REGION Network 8: Reset Counters
   RUNG wire#powerrail
      Contact( #Reset_Counters )
      Move(in := 0, out1 => "DB_STATUS_IJCORE".AW_number)
      Move(in := T#0MS, out1 => "DB_STATUS_IJCORE".AW_durationMax)
   END_RUNG
   // the same network as SCL:
   IF #Reset_Counters THEN
       "DB_STATUS_IJCORE".AW_number := 0;
       "DB_STATUS_IJCORE".AW_durationMax := T#0MS;
   END_IF;
END_REGION
END_FUNCTION_BLOCK

FUNCTION_BLOCK "IJC PROTOCOL"
{ S7_Optimized_Access := 'TRUE' }
AUTHOR : RAUL_ROBINS
VERSION : 0.1
   VAR_INPUT RETAIN
      M_TYPE : String[3];
      M_NBR : DInt;
   END_VAR
   VAR_INPUT 
      DB_REC : DB_ANY;
      DB_SEND : DB_ANY;
      START_MSG : Bool;
      KANBAN : String[30];
      SAP_PN : String[16];
      COMPONENT : String[64];
      START_SCREW : Bool;
      "SCREW T_INT" : Word;
      "SCREW T_FLOAT" : Word;
      "SCREW ANGLE" : Word;
      ERR_RESET : Bool;
      PROCESS_STATUS { ExternalAccessible := 'False'; ExternalVisible := 'False'; ExternalWritable := 'False'} : SInt;
      NUM_OF_PROCESS : SInt;
   END_VAR

   VAR_OUTPUT 
      SEQ_STEP : Int;
      DN : Bool;
      FLT : Bool;
      ANS : SInt;
      A_TMOUT : Bool;
      M_TMOUT : Bool;
      NFP : String[8];
   END_VAR

   VAR_IN_OUT 
      AWAKE_SW : Int;
   END_VAR

   VAR 
      MSG_TMOUT {InstructionName := 'TON_TIME'; LibVersion := '1.0'} : TON_TIME;
      AWK_TMR {InstructionName := 'TON_TIME'; LibVersion := '1.0'} : TON_TIME;
      AWK_TMOUT {InstructionName := 'TON_TIME'; LibVersion := '1.0'} : TON_TIME;
      "SCREW NBR" { S7_SetPoint := 'True'} : Word;
      SCREW : Array[1..9] of Struct
         ANGLE : Word;
         TORQUE : Struct
            "INT" : Word;
            FLOAT : Word;
         END_STRUCT;
      END_STRUCT;
      HMI : Struct
         SEND : Struct
            MSG : String[50];
            SW : SInt;
         END_STRUCT;
         RCV : Struct
            MSG : String[50];
            SW : SInt;
         END_STRUCT;
      END_STRUCT;
      ONS : Array[1..10] of Bool;
   END_VAR

   VAR_TEMP 
      MSG_TYPE : SInt;
      IDB : Int;
      i : Int;
      j : Int;
      k : Int;
      SEND_OFFSET : Struct
         SW : DInt;
         MSG : DInt;
      END_STRUCT;
      REC_OFFSET : Struct
         SW : DInt;
         ANS : DInt;
         MSG : DInt;
      END_STRUCT;
      CNT : SInt;
      CNT_STR : String[2];
      TMP : Word;
      BTEST : Bool;
      STATUS : Char;
      NUMBER : Char;
      CHAR_ARRAY : Array[0..49] of Char;
   END_VAR

   VAR CONSTANT 
      "DB" : Byte := 16#84;
      CLEAR : Word := 16#0;
      MINUS1 : Word := 16#FFFF;
      PLUS1 : Word := 16#1;
   END_VAR


BEGIN
	(*     IJCORE PROTOCOL
	CREATED BY: RAUL ROBINS
	CREATED ON: 08/05/2020
	VERSION: 1.0
	*)
	
	//***** CLEAR ALL FAULTS ***************************************
	IF #ERR_RESET OR
	NOT #START_MSG THEN
	    #M_TMOUT := false;
	    #FLT := FALSE;
	END_IF;
	
	//***** AWAKE SIGNAL ***************************************
	  //#AWK_TMR(IN := (#AWAKE_SW <= 0),
	  //      PT := T#500ms);
	
	//IF #AWK_TMR.Q AND
	  //  #AWAKE_SW <= 1 THEN
	   // #AWAKE_SW := 1;
	//END_IF;
	
	
	//AWAKE TIMEOUT
	//#AWK_TMOUT(IN := (#AWAKE_SW = 1),
	  //      PT := T#6S);
	//IF #AWK_TMOUT.Q THEN
	    //#A_TMOUT := TRUE;
	//ELSIF (#AWAKE_SW < 0) THEN
	  //  #A_TMOUT := FALSE;
	//END_IF;
	
	// ***** TIMEOUT FOR ANSWER FROM IJC **********************************
	// WAITMOUNT FOR FAULT
	// 
	#MSG_TMOUT(IN := (#SEQ_STEP = 50 OR #SEQ_STEP = 60),
	           PT := T#60S,
	           Q => #BTEST);
	//SET FAULT
	 IF #MSG_TMOUT.Q THEN
	     #M_TMOUT := true;
	     #SEQ_STEP := 0;
	END_IF;
	
	//***** VALID MESSAGE NUMBER ***************************************
	IF #M_NBR < 1 THEN
	    RETURN;
	END_IF;
	
	//***** MESSAGE TYPE SELECTED ***************************************
	IF    #M_TYPE = 'CNF' THEN
	    #MSG_TYPE := 1;
	ELSIF #M_TYPE = 'TRC' THEN
	    #MSG_TYPE := 1;
	ELSIF #M_TYPE = 'TRB' THEN
	    #MSG_TYPE := 1;
	ELSIF #M_TYPE = 'TRS' THEN
	    #MSG_TYPE := 2;
	ELSIF #M_TYPE = 'TRI' THEN
	    #MSG_TYPE := 3;
	ELSIF #M_TYPE = 'TRE' THEN
	    #MSG_TYPE := 4;
	ELSIF #M_TYPE = 'STA' THEN
	    #MSG_TYPE := 5;
	ELSIF #M_TYPE = 'CMA' THEN
	    #MSG_TYPE := 6;
	ELSIF #M_TYPE = 'TRR' THEN
	    #MSG_TYPE := 7;
	ELSIF #M_TYPE = 'TRW' THEN
	    #MSG_TYPE := 8;
	ELSIF #M_TYPE = 'PFC' THEN
	    #MSG_TYPE := 9;
	ELSIF #M_TYPE = 'NFP' THEN
	    #MSG_TYPE := 10;
	ELSE
	    RETURN;
	END_IF;
	
	//***** MESSAGE OFFSET CALC ***************************************
	#SEND_OFFSET.SW := (#M_NBR * 2) + 2;
	#SEND_OFFSET.MSG := ((#M_NBR - 1) * 80) + 604;
	#REC_OFFSET.SW := (#M_NBR - 1) * 2;
	#REC_OFFSET.ANS := ((#M_NBR - 1) * 32) + 600;
	#REC_OFFSET.MSG := ((#M_NBR - 1) * 32) + 602;
	#HMI.SEND.SW := WORD_TO_SINT(PEEK_WORD(area := #DB, dbNumber := #DB_SEND, byteOffset := #SEND_OFFSET.SW));
	#HMI.RCV.SW := WORD_TO_SINT(PEEK_WORD(area := #DB, dbNumber := #DB_REC, byteOffset := #REC_OFFSET.SW));
	
	//***** GET SCREW DATA ***************************************
	
	//CLEAR SCREW DATA*************************************************
	// IF NOT #START_SCREW THEN
	//     #"SCREW NBR" := 0;
	//     FOR #i := 1 TO 9 BY 1 DO
	//         #SCREW[#i].TORQUE."INT" := 0;
	//         #SCREW[#i].TORQUE.FLOAT := 0;
	//         #SCREW[#i].ANGLE := 0;
	//     END_FOR;
	// END_IF;
	
	// IF  #START_SCREW   AND
	//     #"SCREW ANGLE" > 0 AND
	//     #"SCREW NBR"< 9 THEN
	//     IF NOT #ONS[2] THEN
	//         #"SCREW NBR" += 1;
	//         #SCREW[#"SCREW NBR"].TORQUE."INT" := #"SCREW T_INT";
	//         #SCREW[#"SCREW NBR"].TORQUE.FLOAT := #"SCREW T_FLOAT";
	//         #SCREW[#"SCREW NBR"].ANGLE := #"SCREW ANGLE";
	// //ONE SHOT
	//         #ONS[2] := True;
	//     END_IF;
	// ELSE
	//     #ONS[2] := False;
	// END_IF;
	#"SCREW NBR" := SINT_TO_WORD(#NUM_OF_PROCESS);
	
	
	////////////////////////////////////////////////////////////////////
	//START IJCORE SEQUENCE
	//>>>>>STEP-00 ->>>>>>>>>>>>>>>>>>>>>>>>>>>>>>>>>>>>>>>>>>>>>>>>>>>>>
	//WAIT FLAG SEND TO START SEQUENCE
	
	IF  NOT #START_MSG THEN
	    #DN := FALSE;
	    #SEQ_STEP := 0;
	    #ANS := 0;
	    //MESSAGE
	    FOR #i := 0 TO 79 DO
	        POKE(area := #DB,
	             dbNumber := #DB_SEND,
	             byteOffset := (#SEND_OFFSET.MSG + #i),
	             value := ' ');
	    END_FOR;
	    //SW_MESSAGE
	    POKE(area := #DB,
	         dbNumber := #DB_SEND,
	         byteOffset := #SEND_OFFSET.SW,
	         value := #CLEAR);
	ELSE
	    //***** HMI SIGNAL STATUS ***************************************
	    //SEND
	    FOR #i := 0 TO 49 BY 1 DO
	        #CHAR_ARRAY[#i] := BYTE_TO_CHAR(PEEK(area := #DB, dbNumber := #DB_SEND, byteOffset := #SEND_OFFSET.MSG + #i));
	    END_FOR;
	    
	    Chars_TO_Strg(Chars := #CHAR_ARRAY,
	                  pChars := 0,
	                  Cnt := 50,
	                  Strg => #HMI.SEND.MSG);
	    
	    
	    //NFP
	    //
	    
	    // #NFP := '';
	
	    // RETURN;
	END_IF;
	
	
	//***** HMI SIGNAL STATUS ***************************************
	//SEND
	//FOR #i := 0 TO 49 BY 1 DO
	  //  #CHAR_ARRAY[#i] := BYTE_TO_CHAR(PEEK(area := #DB, dbNumber := #DB_SEND, byteOffset := #SEND_OFFSET.MSG + #i));
	//END_FOR;
	
	//Chars_TO_Strg(Chars := #CHAR_ARRAY,
	  //            pChars := 0,
	    //          #CNT := 50,
	      //        Strg => #HMI.SEND.MSG);
	
	
	//HMI REC
	FOR #i := 0 TO 49 BY 1 DO
	    #CHAR_ARRAY[#i] := BYTE_TO_CHAR(PEEK(area := #DB, dbNumber := #DB_REC, byteOffset := #REC_OFFSET.MSG + #i));
	END_FOR;
	
	Chars_TO_Strg(Chars := #CHAR_ARRAY,
	              pChars := 0,
	              Cnt := 50,
	              Strg => #HMI.RCV.MSG);
	
	//***** START SEQUENCE ***************************************
	IF #SEQ_STEP = 0 AND #SEQ_STEP<>100 AND 
	    #START_MSG THEN
	    #SEQ_STEP := 10;
	END_IF;
	
	//>>>>>STEP-10 ->>>>>>>>>>>>>>>>>>>>>>>>>>>>>>>>>>>>>>>>>>>>>>>>>>>>>
	//TURN OFF SEND FLAG
	IF #SEQ_STEP = 10 AND #SEQ_STEP<>100 AND  #START_MSG THEN
	    //GOTO STEP 30
	    #SEQ_STEP := 30;
	END_IF;
	
	//>>>>>STEP-30 ->>>>>>>>>>>>>>>>>>>>>>>>>>>>>>>>>>>>>>>>>>>>>>>>>>>>>
	//INIT DATA DB5 or DB1005 
	IF #SEQ_STEP = 30 THEN
	    //SET FLAGS TO 0
	    POKE(area := #DB,
	         dbNumber := #DB_SEND,
	         byteOffset := #SEND_OFFSET.SW,
	         value := #CLEAR);
	    POKE(area := #DB,
	         dbNumber := #DB_REC,
	         byteOffset := #REC_OFFSET.SW,
	         value := #CLEAR);
	    POKE(area := #DB,
	         dbNumber := #DB_REC,
	         byteOffset := #REC_OFFSET.ANS,
	         value := #CLEAR);
	    
	    //CLEAR DBSEND MESSAGE
	    FOR #i := 0 TO 79 BY 1 DO
	        POKE(area := #DB,
	             dbNumber := #DB_SEND,
	             byteOffset := (#SEND_OFFSET.MSG + #i),
	             value := ' ');
	    END_FOR;
	    FOR #i := 0 TO 69 BY 1 DO
	        POKE(area := #DB,
	             dbNumber := #DB_REC,
	             byteOffset := (#REC_OFFSET.MSG + #i),
	             value := ' ');
	    END_FOR;
	    //GO TO STEP 40
	    #SEQ_STEP := 40;
	END_IF;
	
	//>>>>>STEP-40 ->>>>>>>>>>>>>>>>>>>>>>>>>>>>>>>>>>>>>>>>>>>>>>>>>>>>>
	//CREATE MESSAGE
	IF #SEQ_STEP = 40 THEN
	    //MESSAGE TYPE
	   
	    //COPY KANBAN
	    FOR #i := 0 TO 7 BY 1 DO
	        POKE(area := #DB,
	             dbNumber := #DB_SEND,
	             byteOffset := (#SEND_OFFSET.MSG + #i),
	             value := #KANBAN[#i+1]);
	    END_FOR;
	    
	    //CONVERT DATATYPE
	    #STATUS := SINT_TO_CHAR(#PROCESS_STATUS + 48);
	    #NUMBER := SINT_TO_CHAR(#NUM_OF_PROCESS + 48);
	    
	    CASE #MSG_TYPE OF
	        1://CNF & TRC
	            #CNT := INT_TO_SINT (LEN(#COMPONENT));
	            VAL_STRG(IN := #CNT,
	                     SIZE := 2,
	                     PREC := 0,
	                     FORMAT := W#16#0,
	                     P := 1,
	                     OUT => #CNT_STR);
	            IF #CNT < 10 THEN
	                #CNT_STR := REPLACE(IN1 := #CNT_STR, IN2 := '0',
	                                    L := 1,
	                                    P := FIND(IN1 := #CNT_STR,
	                                              IN2 := ' '));
	            END_IF;
	            POKE(area := #DB,
	                 dbNumber := #DB_SEND,
	                 byteOffset := (#SEND_OFFSET.MSG + 8),
	                 value := #CNT_STR[1]);
	            POKE(area := #DB,
	                 dbNumber := #DB_SEND,
	                 byteOffset := (#SEND_OFFSET.MSG + 9),
	                 value := #CNT_STR[2]);
	            FOR #i := 0 TO 28 BY 1 DO
	                POKE(area := #DB,
	                     dbNumber := #DB_SEND,
	                     byteOffset := (#SEND_OFFSET.MSG + #i + 10),
	                     value := #COMPONENT[#i+1]);
	            END_FOR;
	            
	        2://TRS
	            #NUMBER := WORD_TO_CHAR(#"SCREW NBR" + 48);
	            POKE(area := #DB,
	                 dbNumber := #DB_SEND,
	                 byteOffset := (#SEND_OFFSET.MSG + 8),
	                 value := #STATUS);
	            POKE(area := #DB,
	                 dbNumber := #DB_SEND,
	                 byteOffset := (#SEND_OFFSET.MSG + 9),
	                 value := #NUMBER);
	            FOR #i := 0 TO 8 BY 1 DO
	                #j := #i + 1;
	                #k := (#i * 6) + 10;
	                //ANGLE
	                POKE(area := #DB,
	                     dbNumber := #DB_SEND,
	                     byteOffset := (#SEND_OFFSET.MSG + #k ),
	                     value :=  #SCREW[#j].ANGLE);
	                //TORQUE BEFORE POINT
	                POKE(area := #DB,
	                     dbNumber := #DB_SEND,
	                     byteOffset := (#SEND_OFFSET.MSG + #k + 2),
	                     value := #SCREW[#j].TORQUE."INT");
	        
	                //TORQUE AFTER POINT
	                POKE(area := #DB,
	                     dbNumber := #DB_SEND,
	                     byteOffset := (#SEND_OFFSET.MSG + #k + 4),
	                     value := #SCREW[#j].TORQUE."FLOAT");
	            END_FOR;
	            
	        3://TRI
	            POKE(area := #DB,
	                 dbNumber := #DB_SEND,
	                 byteOffset := (#SEND_OFFSET.MSG + 8),
	                 value := #STATUS);
	        4://TRE 
	            POKE(area := #DB,
	                 dbNumber := #DB_SEND,
	                 byteOffset := (#SEND_OFFSET.MSG + 8),
	                 value := '9');;
	            POKE(area := #DB,
	                 dbNumber := #DB_SEND,
	                 byteOffset := (#SEND_OFFSET.MSG + 9),     
	                 value := '9');                                 
	            POKE(area := #DB,
	                 dbNumber := #DB_SEND,
	                 byteOffset := (#SEND_OFFSET.MSG + 10),
	                 value := #STATUS);
	        5://STA
	            ;
	        6://TRB
	            POKE(area := #DB,
	                 dbNumber := #DB_SEND,
	                 byteOffset := (#SEND_OFFSET.MSG + 9),
	                 value := '1');;
	            POKE(area := #DB,
	                 dbNumber := #DB_SEND,
	                 byteOffset := (#SEND_OFFSET.MSG + 10),
	                 value := '6');
	            FOR #i := 1 TO 16 BY 1 DO
	                POKE(area := #DB,
	                     dbNumber := #DB_SEND,
	                     byteOffset := (#SEND_OFFSET.MSG + #i + 1),
	                     value := #SAP_PN[#i]);
	            END_FOR;
	            ;
	        7://TRR
	            POKE(area := #DB,
	                 dbNumber := #DB_SEND,
	                 byteOffset := (#SEND_OFFSET.MSG + 8),
	                 value := #STATUS);
	            POKE(area := #DB,
	                 dbNumber := #DB_SEND,
	                 byteOffset := (#SEND_OFFSET.MSG + 9),
	                 value := #NUMBER);
	            
	        8://TRW
	            POKE(area := #DB,
	                 dbNumber := #DB_SEND,
	                 byteOffset := (#SEND_OFFSET.MSG + 8),
	                 value := #STATUS);
	            POKE(area := #DB,
	                 dbNumber := #DB_SEND,
	                 byteOffset := (#SEND_OFFSET.MSG + 9),
	                 value := #NUMBER);
	            
	        9://PFC
	            #CNT := INT_TO_SINT(LEN(#COMPONENT));
	            VAL_STRG(IN := #CNT,
	                     SIZE := 2,
	                     PREC := 0,
	                     FORMAT := W#16#0,
	                     P := 1,
	                     OUT => #CNT_STR);
	            IF #CNT < 10 THEN
	                #CNT_STR := REPLACE(IN1 := #CNT_STR, IN2 := '0',
	                                    L := 1,
	                                    P := FIND(IN1 := #CNT_STR,
	                                              IN2 := ' '));
	            END_IF;
	            POKE(area := #DB,
	                 dbNumber := #DB_SEND,
	                 byteOffset := (#SEND_OFFSET.MSG + 8),
	                 value := #CNT_STR[1]);
	            POKE(area := #DB,
	                 dbNumber := #DB_SEND,
	                 byteOffset := (#SEND_OFFSET.MSG + 9),
	                 value := #CNT_STR[2]);
	            FOR #i := 0 TO 28 BY 1 DO
	                POKE(area := #DB,
	                     dbNumber := #DB_SEND,
	                     byteOffset := (#SEND_OFFSET.MSG + #i + 10),
	                     value := #COMPONENT[#i + 1]);
	            END_FOR;
	        10://NFP
	            POKE(area := #DB,
	                 dbNumber := #DB_SEND,
	                 byteOffset := (#SEND_OFFSET.MSG),
	                 value := '0');
	            POKE(area := #DB,
	                 dbNumber := #DB_SEND,
	                 byteOffset := (#SEND_OFFSET.MSG + 1),
	                 value := '8');
	            FOR #i := 1 TO 8 BY 1 DO
	                POKE(area := #DB,
	                     dbNumber := #DB_SEND,
	                     byteOffset := (#SEND_OFFSET.MSG + #i + 1),
	                     value := #KANBAN[#i]);
	            END_FOR;
	    END_CASE;
	    
	    //SET FLAG TO I TO INFORM THAT PLC IS READY (DB5 Ó 1005)
	    POKE(area := #DB,
	         dbNumber := #DB_SEND,
	         byteOffset := #SEND_OFFSET.SW,
	         value := #PLUS1);
	   #SEQ_STEP := 50;
	END_IF;
	
	//***** WAIT ANSWER FROM IJC***** **********************************
	//CHECK FLAG IN STEP-50
	IF #SEQ_STEP = 50 THEN
	    //WAIT FOR SEND FLAG TO BE -1
	    IF PEEK_WORD(area := #DB, dbNumber := #DB_SEND, byteOffset := #SEND_OFFSET.SW) = #MINUS1 THEN
	        #SEQ_STEP := 60;//GO TO STEP 60
	    END_IF;
	END_IF;
	
	//>>>>>STEP-60 ->>>>>>>>>>>>>>>>>>>>>>>>>>>>>>>>>>>>>>>>>>>>>>>>>>>>>
	//COPY NFP MESSAGE TO LOCAL IJC_DB AND ANSWER -1 TO IJC
	IF #SEQ_STEP = 60 THEN
	    //POINTER OFFSET TO STATUS WORD
	    IF PEEK_WORD(area := #DB, dbNumber := #DB_REC, byteOffset := #REC_OFFSET.SW) = #PLUS1 THEN
	        #ANS := (PEEK_WORD(area := #DB, dbNumber := #DB_REC, byteOffset := #REC_OFFSET.ANS));
	        #TMP := (PEEK_WORD(area := #DB, dbNumber := #DB_REC, byteOffset := #REC_OFFSET.ANS));
	     //COPY NFP RECEIVED
	        FOR #i := 0 TO 7 BY 1 DO
	            #CHAR_ARRAY[#i] := PEEK_BYTE(area := #DB, dbNumber := #DB_REC, byteOffset := #REC_OFFSET.MSG+#i);
	        END_FOR;
	        Chars_TO_Strg(Chars:=#CHAR_ARRAY,
	                      pChars:=0,
	                      Cnt:=8,
	                      Strg=>#NFP);
	        //SET TO -1 REC
	        POKE(area := #DB,
	             dbNumber := #DB_REC,
	             byteOffset := #REC_OFFSET.SW,
	             value := #MINUS1);
	        #DN := TRUE;
	        #SEQ_STEP := 100;
	    END_IF;
	END_IF;
	
	
	IF #TMP < 0 THEN
	    #FLT := TRUE;
	END_IF;
	//RESET FAULT
	
	
	//***** END**********************************************************************
	
END_FUNCTION_BLOCK

FUNCTION_BLOCK "IJCoreMain"   // FB1000, LAD
TITLE = IJCore Main
{ S7_Optimized_Access := 'TRUE' }
VERSION : 0.1
// stored: AutoNumber false, IsIECCheckEnabled false, IsRetainMemResEnabled false, MemoryReserve 100, SetENOAutomatically false, UDAEnableTagReadback false
   VAR
      Enable : Bool;
      Mode : UInt;
      Indicator : Int;
      AlarmReset : Bool;
      AWAKE_SIGNAL { S7_SetPoint := 'True'} : "AWAKE_SIGNAL";
      MSG : Array[1..20] of "IJCoreMessageProcotol";
      NFP { S7_SetPoint := 'True'} : Array[1..4] of String[30];
   END_VAR
   VAR_TEMP
      MessageDone : Bool;
      Answer : DInt;
      Fault : DInt;
   END_VAR
   VAR CONSTANT
      STA : Int := 5;
      CNF : Int := 1;
      TRC : Int := 13;
      PFC : Int := 9;
      TRR : Int := 7;
   END_VAR
BEGIN

REGION Network 1
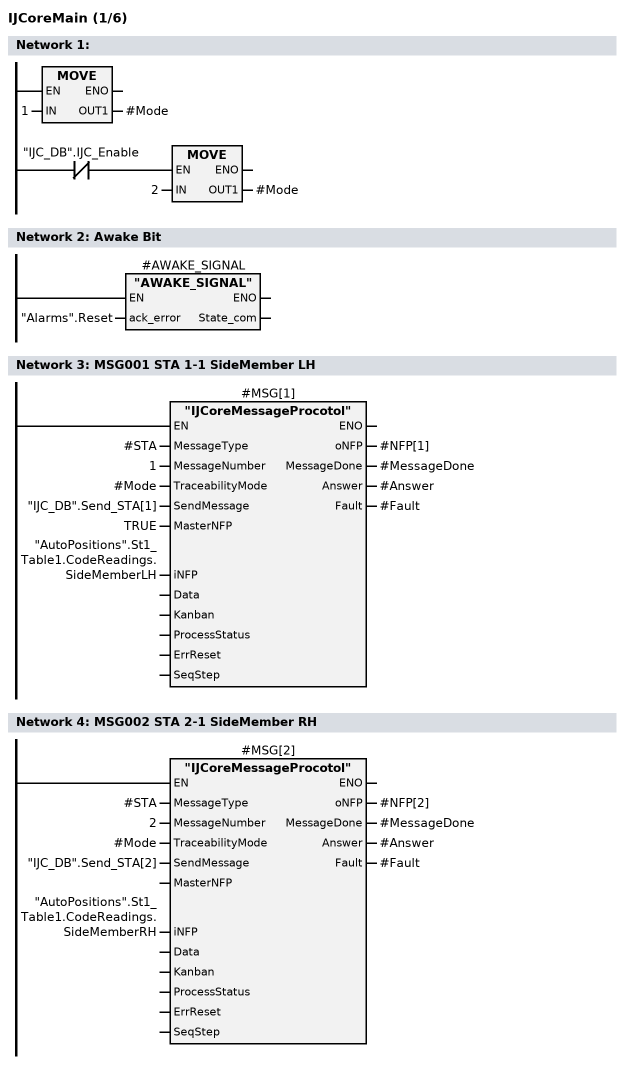
   RUNG wire#powerrail
      Move(in := 1, out1 => #Mode)
   END_RUNG
   RUNG wire#powerrail
      I_Contact( "IJC_DB".IJC_Enable )
      Move(in := 2, out1 => #Mode)
   END_RUNG
   // the same network as SCL:
   #Mode := 1;
   IF NOT "IJC_DB".IJC_Enable THEN #Mode := 2; END_IF;
END_REGION

REGION Network 2: Awake Bit
   RUNG wire#powerrail
      #AWAKE_SIGNAL(ack_error := "Alarms".Reset, State_com =>)
   END_RUNG
   // the same network as SCL:
   #AWAKE_SIGNAL(ack_error := "Alarms".Reset);   // "AWAKE_SIGNAL"
END_REGION

REGION Network 3: MSG001 STA 1-1 SideMember LH
   RUNG wire#powerrail
      #MSG[1](MessageType := #STA, MessageNumber := 1, TraceabilityMode := #Mode, SendMessage := "IJC_DB".Send_STA[1], MasterNFP := TRUE, iNFP := "AutoPositions".St1_Table1.CodeReadings.SideMemberLH, Data :=, Kanban :=, ProcessStatus :=, ErrReset :=, SeqStep :=, oNFP => #NFP[1], MessageDone => #MessageDone, Answer => #Answer, Fault => #Fault)
   END_RUNG
   // the same network as SCL:
   #MSG[1](MessageType := #STA,   // "IJCoreMessageProcotol"
           MessageNumber := 1,
           TraceabilityMode := #Mode,
           SendMessage := "IJC_DB".Send_STA[1],
           MasterNFP := TRUE,
           iNFP := "AutoPositions".St1_Table1.CodeReadings.SideMemberLH,
           oNFP => #NFP[1],
           MessageDone => #MessageDone,
           Answer => #Answer,
           Fault => #Fault);
END_REGION

REGION Network 4: MSG002 STA 2-1 SideMember RH
   RUNG wire#powerrail
      #MSG[2](MessageType := #STA, MessageNumber := 2, TraceabilityMode := #Mode, SendMessage := "IJC_DB".Send_STA[2], MasterNFP :=, iNFP := "AutoPositions".St1_Table1.CodeReadings.SideMemberRH, Data :=, Kanban :=, ProcessStatus :=, ErrReset :=, SeqStep :=, oNFP => #NFP[2], MessageDone => #MessageDone, Answer => #Answer, Fault => #Fault)
   END_RUNG
   // the same network as SCL:
   #MSG[2](MessageType := #STA,   // "IJCoreMessageProcotol"
           MessageNumber := 2,
           TraceabilityMode := #Mode,
           SendMessage := "IJC_DB".Send_STA[2],
           iNFP := "AutoPositions".St1_Table1.CodeReadings.SideMemberRH,
           oNFP => #NFP[2],
           MessageDone => #MessageDone,
           Answer => #Answer,
           Fault => #Fault);
END_REGION

REGION Network 5: MSG003 STA 3-1 Front Tube
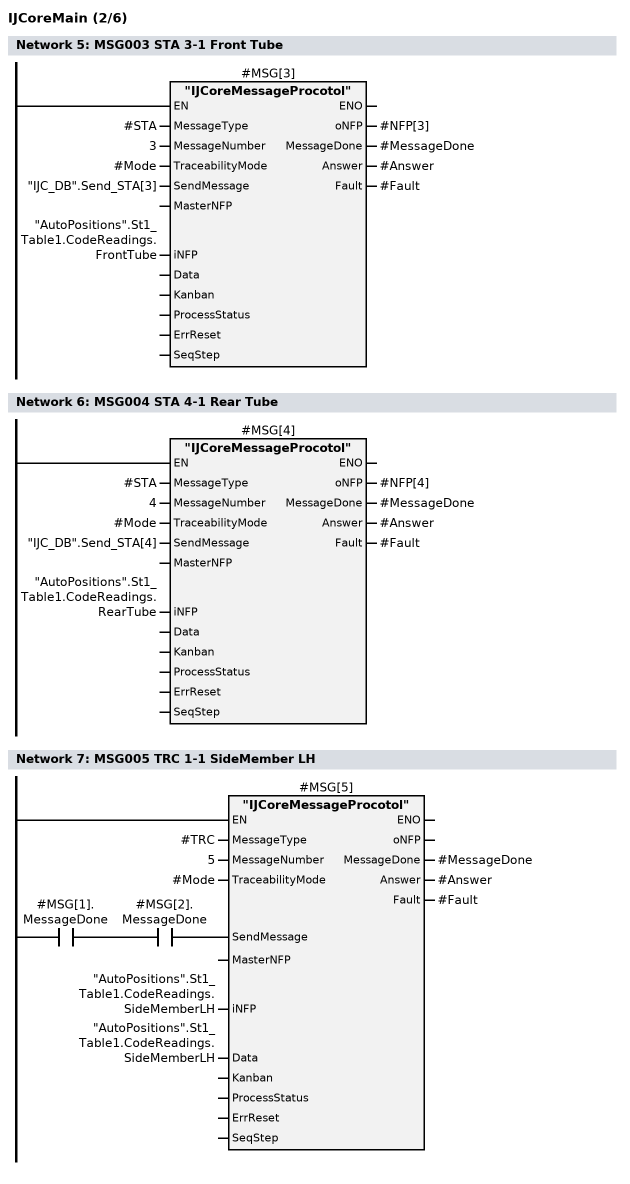
   RUNG wire#powerrail
      #MSG[3](MessageType := #STA, MessageNumber := 3, TraceabilityMode := #Mode, SendMessage := "IJC_DB".Send_STA[3], MasterNFP :=, iNFP := "AutoPositions".St1_Table1.CodeReadings.FrontTube, Data :=, Kanban :=, ProcessStatus :=, ErrReset :=, SeqStep :=, oNFP => #NFP[3], MessageDone => #MessageDone, Answer => #Answer, Fault => #Fault)
   END_RUNG
   // the same network as SCL:
   #MSG[3](MessageType := #STA,   // "IJCoreMessageProcotol"
           MessageNumber := 3,
           TraceabilityMode := #Mode,
           SendMessage := "IJC_DB".Send_STA[3],
           iNFP := "AutoPositions".St1_Table1.CodeReadings.FrontTube,
           oNFP => #NFP[3],
           MessageDone => #MessageDone,
           Answer => #Answer,
           Fault => #Fault);
END_REGION

REGION Network 6: MSG004 STA 4-1 Rear Tube
   RUNG wire#powerrail
      #MSG[4](MessageType := #STA, MessageNumber := 4, TraceabilityMode := #Mode, SendMessage := "IJC_DB".Send_STA[4], MasterNFP :=, iNFP := "AutoPositions".St1_Table1.CodeReadings.RearTube, Data :=, Kanban :=, ProcessStatus :=, ErrReset :=, SeqStep :=, oNFP => #NFP[4], MessageDone => #MessageDone, Answer => #Answer, Fault => #Fault)
   END_RUNG
   // the same network as SCL:
   #MSG[4](MessageType := #STA,   // "IJCoreMessageProcotol"
           MessageNumber := 4,
           TraceabilityMode := #Mode,
           SendMessage := "IJC_DB".Send_STA[4],
           iNFP := "AutoPositions".St1_Table1.CodeReadings.RearTube,
           oNFP => #NFP[4],
           MessageDone => #MessageDone,
           Answer => #Answer,
           Fault => #Fault);
END_REGION

REGION Network 7: MSG005 TRC 1-1 SideMember LH
   RUNG wire#powerrail
      #MSG[5](SendMessage := wire#w1, MessageType := #TRC, MessageNumber := 5, TraceabilityMode := #Mode, MasterNFP :=, iNFP := "AutoPositions".St1_Table1.CodeReadings.SideMemberLH, Data := "AutoPositions".St1_Table1.CodeReadings.SideMemberLH, Kanban :=, ProcessStatus :=, ErrReset :=, SeqStep :=, oNFP =>, MessageDone => #MessageDone, Answer => #Answer, Fault => #Fault)
   END_RUNG
   RUNG wire#powerrail
      Contact( #MSG[1].MessageDone )
      Contact( #MSG[2].MessageDone )
   END_RUNG wire#w1
   // the same network as SCL:
   #MSG[5](MessageType := #TRC,   // "IJCoreMessageProcotol"
           MessageNumber := 5,
           TraceabilityMode := #Mode,
           SendMessage := #MSG[1].MessageDone AND #MSG[2].MessageDone,
           iNFP := "AutoPositions".St1_Table1.CodeReadings.SideMemberLH,
           Data := "AutoPositions".St1_Table1.CodeReadings.SideMemberLH,
           MessageDone => #MessageDone,
           Answer => #Answer,
           Fault => #Fault);
END_REGION

REGION Network 8: MSG006 TRC 1-2 SideMember RH
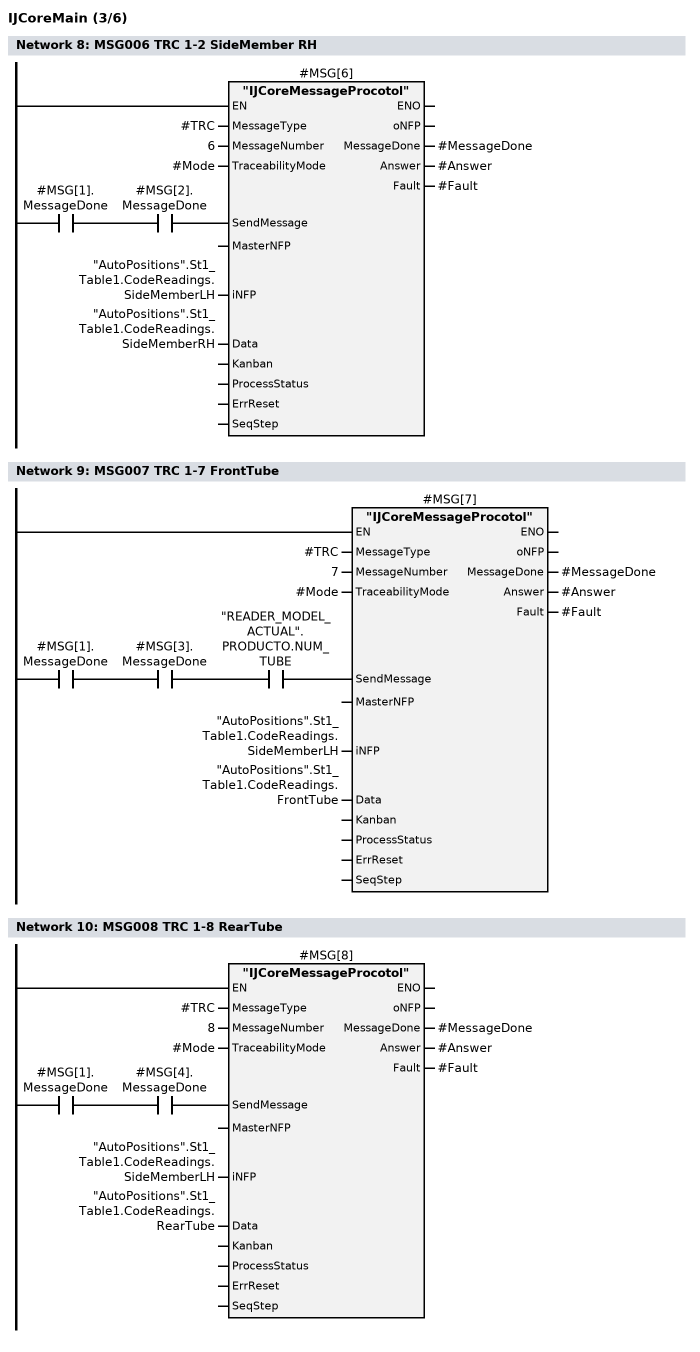
   RUNG wire#powerrail
      #MSG[6](SendMessage := wire#w1, MessageType := #TRC, MessageNumber := 6, TraceabilityMode := #Mode, MasterNFP :=, iNFP := "AutoPositions".St1_Table1.CodeReadings.SideMemberLH, Data := "AutoPositions".St1_Table1.CodeReadings.SideMemberRH, Kanban :=, ProcessStatus :=, ErrReset :=, SeqStep :=, oNFP =>, MessageDone => #MessageDone, Answer => #Answer, Fault => #Fault)
   END_RUNG
   RUNG wire#powerrail
      Contact( #MSG[1].MessageDone )
      Contact( #MSG[2].MessageDone )
   END_RUNG wire#w1
   // the same network as SCL:
   #MSG[6](MessageType := #TRC,   // "IJCoreMessageProcotol"
           MessageNumber := 6,
           TraceabilityMode := #Mode,
           SendMessage := #MSG[1].MessageDone AND #MSG[2].MessageDone,
           iNFP := "AutoPositions".St1_Table1.CodeReadings.SideMemberLH,
           Data := "AutoPositions".St1_Table1.CodeReadings.SideMemberRH,
           MessageDone => #MessageDone,
           Answer => #Answer,
           Fault => #Fault);
END_REGION

REGION Network 9: MSG007 TRC 1-7 FrontTube
   RUNG wire#powerrail
      #MSG[7](SendMessage := wire#w1, MessageType := #TRC, MessageNumber := 7, TraceabilityMode := #Mode, MasterNFP :=, iNFP := "AutoPositions".St1_Table1.CodeReadings.SideMemberLH, Data := "AutoPositions".St1_Table1.CodeReadings.FrontTube, Kanban :=, ProcessStatus :=, ErrReset :=, SeqStep :=, oNFP =>, MessageDone => #MessageDone, Answer => #Answer, Fault => #Fault)
   END_RUNG
   RUNG wire#powerrail
      Contact( #MSG[1].MessageDone )
      Contact( #MSG[3].MessageDone )
      Contact( "READER_MODEL_ACTUAL".PRODUCTO.NUM_TUBE )
   END_RUNG wire#w1
   // the same network as SCL:
   #MSG[7](MessageType := #TRC,   // "IJCoreMessageProcotol"
           MessageNumber := 7,
           TraceabilityMode := #Mode,
           SendMessage := #MSG[1].MessageDone AND #MSG[3].MessageDone AND "READER_MODEL_ACTUAL".PRODUCTO.NUM_TUBE,
           iNFP := "AutoPositions".St1_Table1.CodeReadings.SideMemberLH,
           Data := "AutoPositions".St1_Table1.CodeReadings.FrontTube,
           MessageDone => #MessageDone,
           Answer => #Answer,
           Fault => #Fault);
END_REGION

REGION Network 10: MSG008 TRC 1-8 RearTube
   RUNG wire#powerrail
      #MSG[8](SendMessage := wire#w1, MessageType := #TRC, MessageNumber := 8, TraceabilityMode := #Mode, MasterNFP :=, iNFP := "AutoPositions".St1_Table1.CodeReadings.SideMemberLH, Data := "AutoPositions".St1_Table1.CodeReadings.RearTube, Kanban :=, ProcessStatus :=, ErrReset :=, SeqStep :=, oNFP =>, MessageDone => #MessageDone, Answer => #Answer, Fault => #Fault)
   END_RUNG
   RUNG wire#powerrail
      Contact( #MSG[1].MessageDone )
      Contact( #MSG[4].MessageDone )
   END_RUNG wire#w1
   // the same network as SCL:
   #MSG[8](MessageType := #TRC,   // "IJCoreMessageProcotol"
           MessageNumber := 8,
           TraceabilityMode := #Mode,
           SendMessage := #MSG[1].MessageDone AND #MSG[4].MessageDone,
           iNFP := "AutoPositions".St1_Table1.CodeReadings.SideMemberLH,
           Data := "AutoPositions".St1_Table1.CodeReadings.RearTube,
           MessageDone => #MessageDone,
           Answer => #Answer,
           Fault => #Fault);
END_REGION

REGION Network 11: MSG009 TRR 1-1 Results of riveting
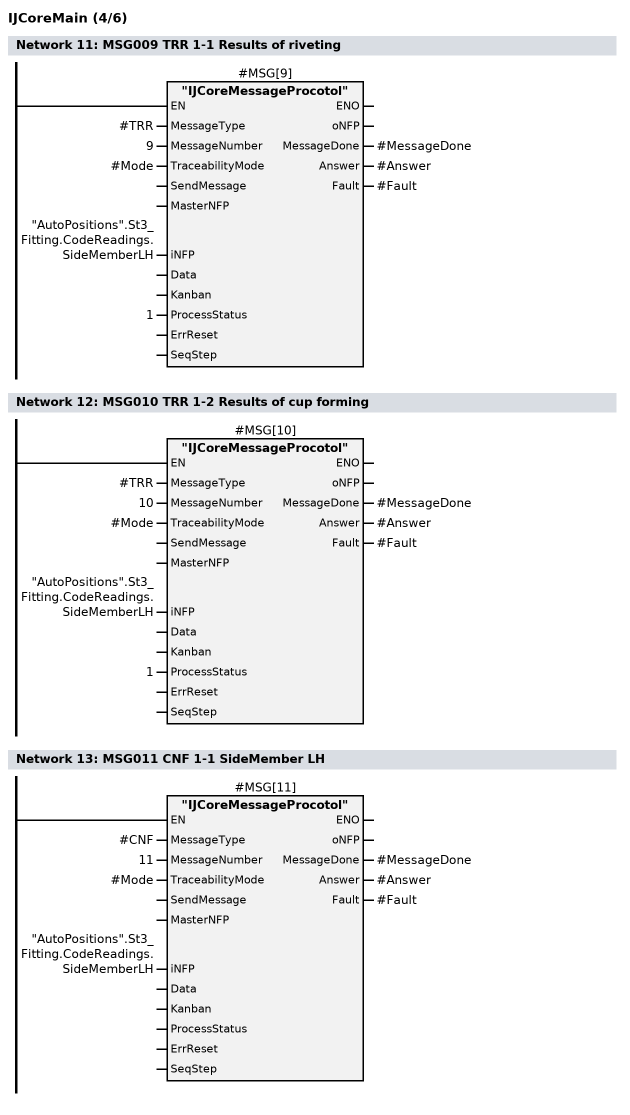
   RUNG wire#powerrail
      #MSG[9](MessageType := #TRR, MessageNumber := 9, TraceabilityMode := #Mode, SendMessage :=, MasterNFP :=, iNFP := "AutoPositions".St3_Fitting.CodeReadings.SideMemberLH, Data :=, Kanban :=, ProcessStatus := 1, ErrReset :=, SeqStep :=, oNFP =>, MessageDone => #MessageDone, Answer => #Answer, Fault => #Fault)
   END_RUNG
   // the same network as SCL:
   #MSG[9](MessageType := #TRR,   // "IJCoreMessageProcotol"
           MessageNumber := 9,
           TraceabilityMode := #Mode,
           iNFP := "AutoPositions".St3_Fitting.CodeReadings.SideMemberLH,
           ProcessStatus := 1,
           MessageDone => #MessageDone,
           Answer => #Answer,
           Fault => #Fault);
END_REGION

REGION Network 12: MSG010 TRR 1-2 Results of cup forming
   RUNG wire#powerrail
      #MSG[10](MessageType := #TRR, MessageNumber := 10, TraceabilityMode := #Mode, SendMessage :=, MasterNFP :=, iNFP := "AutoPositions".St3_Fitting.CodeReadings.SideMemberLH, Data :=, Kanban :=, ProcessStatus := 1, ErrReset :=, SeqStep :=, oNFP =>, MessageDone => #MessageDone, Answer => #Answer, Fault => #Fault)
   END_RUNG
   // the same network as SCL:
   #MSG[10](MessageType := #TRR,   // "IJCoreMessageProcotol"
            MessageNumber := 10,
            TraceabilityMode := #Mode,
            iNFP := "AutoPositions".St3_Fitting.CodeReadings.SideMemberLH,
            ProcessStatus := 1,
            MessageDone => #MessageDone,
            Answer => #Answer,
            Fault => #Fault);
END_REGION

REGION Network 13: MSG011 CNF 1-1 SideMember LH
   RUNG wire#powerrail
      #MSG[11](MessageType := #CNF, MessageNumber := 11, TraceabilityMode := #Mode, SendMessage :=, MasterNFP :=, iNFP := "AutoPositions".St3_Fitting.CodeReadings.SideMemberLH, Data :=, Kanban :=, ProcessStatus :=, ErrReset :=, SeqStep :=, oNFP =>, MessageDone => #MessageDone, Answer => #Answer, Fault => #Fault)
   END_RUNG
   // the same network as SCL:
   #MSG[11](MessageType := #CNF,   // "IJCoreMessageProcotol"
            MessageNumber := 11,
            TraceabilityMode := #Mode,
            iNFP := "AutoPositions".St3_Fitting.CodeReadings.SideMemberLH,
            MessageDone => #MessageDone,
            Answer => #Answer,
            Fault => #Fault);
END_REGION

REGION Network 14: MSG012 CNF 1-2 SideMember RH
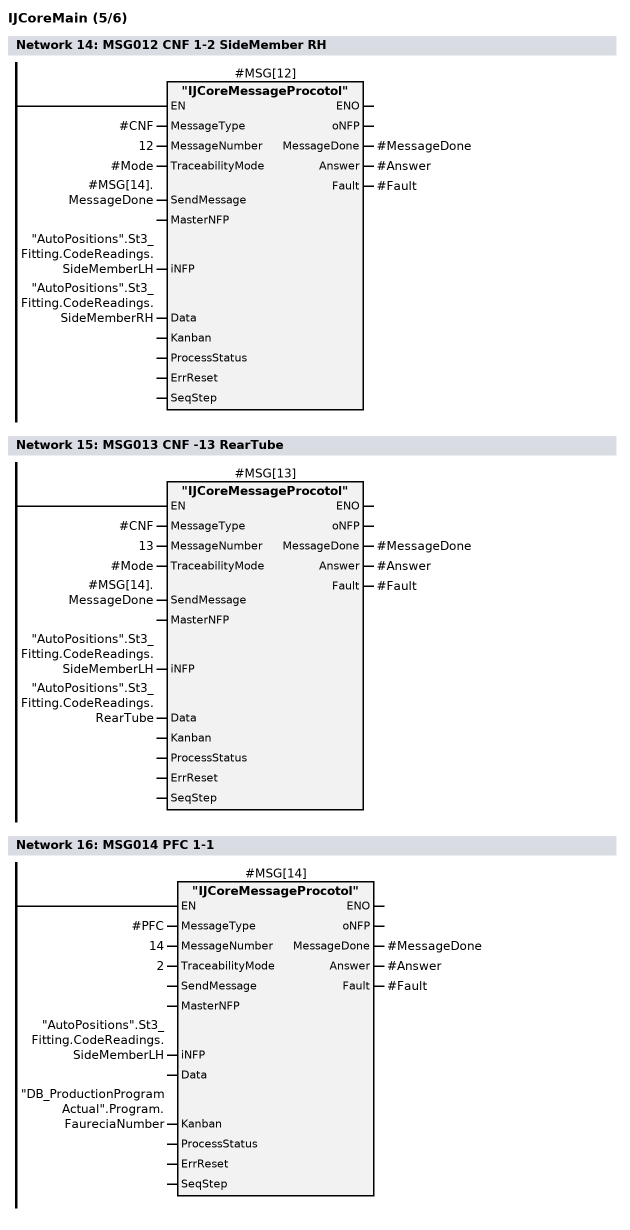
   RUNG wire#powerrail
      #MSG[12](MessageType := #CNF, MessageNumber := 12, TraceabilityMode := #Mode, SendMessage := #MSG[14].MessageDone, MasterNFP :=, iNFP := "AutoPositions".St3_Fitting.CodeReadings.SideMemberLH, Data := "AutoPositions".St3_Fitting.CodeReadings.SideMemberRH, Kanban :=, ProcessStatus :=, ErrReset :=, SeqStep :=, oNFP =>, MessageDone => #MessageDone, Answer => #Answer, Fault => #Fault)
   END_RUNG
   // the same network as SCL:
   #MSG[12](MessageType := #CNF,   // "IJCoreMessageProcotol"
            MessageNumber := 12,
            TraceabilityMode := #Mode,
            SendMessage := #MSG[14].MessageDone,
            iNFP := "AutoPositions".St3_Fitting.CodeReadings.SideMemberLH,
            Data := "AutoPositions".St3_Fitting.CodeReadings.SideMemberRH,
            MessageDone => #MessageDone,
            Answer => #Answer,
            Fault => #Fault);
END_REGION

REGION Network 15: MSG013 CNF -13 RearTube
   RUNG wire#powerrail
      #MSG[13](MessageType := #CNF, MessageNumber := 13, TraceabilityMode := #Mode, SendMessage := #MSG[14].MessageDone, MasterNFP :=, iNFP := "AutoPositions".St3_Fitting.CodeReadings.SideMemberLH, Data := "AutoPositions".St3_Fitting.CodeReadings.RearTube, Kanban :=, ProcessStatus :=, ErrReset :=, SeqStep :=, oNFP =>, MessageDone => #MessageDone, Answer => #Answer, Fault => #Fault)
   END_RUNG
   // the same network as SCL:
   #MSG[13](MessageType := #CNF,   // "IJCoreMessageProcotol"
            MessageNumber := 13,
            TraceabilityMode := #Mode,
            SendMessage := #MSG[14].MessageDone,
            iNFP := "AutoPositions".St3_Fitting.CodeReadings.SideMemberLH,
            Data := "AutoPositions".St3_Fitting.CodeReadings.RearTube,
            MessageDone => #MessageDone,
            Answer => #Answer,
            Fault => #Fault);
END_REGION

REGION Network 16: MSG014 PFC 1-1
   RUNG wire#powerrail
      #MSG[14](MessageType := #PFC, MessageNumber := 14, TraceabilityMode := 2, SendMessage :=, MasterNFP :=, iNFP := "AutoPositions".St3_Fitting.CodeReadings.SideMemberLH, Data :=, Kanban := "DB_ProductionProgramActual".Program.FaureciaNumber, ProcessStatus :=, ErrReset :=, SeqStep :=, oNFP =>, MessageDone => #MessageDone, Answer => #Answer, Fault => #Fault)
   END_RUNG
   // the same network as SCL:
   #MSG[14](MessageType := #PFC,   // "IJCoreMessageProcotol"
            MessageNumber := 14,
            TraceabilityMode := 2,
            iNFP := "AutoPositions".St3_Fitting.CodeReadings.SideMemberLH,
            Kanban := "DB_ProductionProgramActual".Program.FaureciaNumber,
            MessageDone => #MessageDone,
            Answer => #Answer,
            Fault => #Fault);
END_REGION

REGION Network 17: MSG015 CNF 1-4 Front Tube
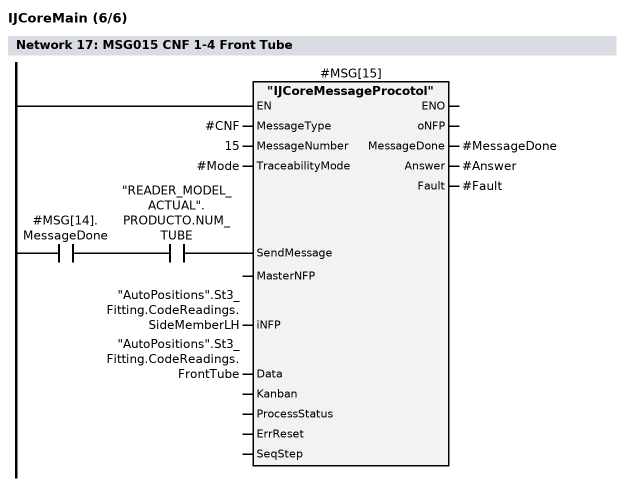
   RUNG wire#powerrail
      #MSG[15](SendMessage := wire#w1, MessageType := #CNF, MessageNumber := 15, TraceabilityMode := #Mode, MasterNFP :=, iNFP := "AutoPositions".St3_Fitting.CodeReadings.SideMemberLH, Data := "AutoPositions".St3_Fitting.CodeReadings.FrontTube, Kanban :=, ProcessStatus :=, ErrReset :=, SeqStep :=, oNFP =>, MessageDone => #MessageDone, Answer => #Answer, Fault => #Fault)
   END_RUNG
   RUNG wire#powerrail
      Contact( #MSG[14].MessageDone )
      Contact( "READER_MODEL_ACTUAL".PRODUCTO.NUM_TUBE )
   END_RUNG wire#w1
   // the same network as SCL:
   #MSG[15](MessageType := #CNF,   // "IJCoreMessageProcotol"
            MessageNumber := 15,
            TraceabilityMode := #Mode,
            SendMessage := #MSG[14].MessageDone AND "READER_MODEL_ACTUAL".PRODUCTO.NUM_TUBE,
            iNFP := "AutoPositions".St3_Fitting.CodeReadings.SideMemberLH,
            Data := "AutoPositions".St3_Fitting.CodeReadings.FrontTube,
            MessageDone => #MessageDone,
            Answer => #Answer,
            Fault => #Fault);
END_REGION
END_FUNCTION_BLOCK

ORGANIZATION_BLOCK "Startup"   // OB124, LAD, Startup
TITLE = "Complete Restart"
{ S7_Optimized_Access := 'TRUE' }
VERSION : 0.1
// stored: AutoNumber true, IsIECCheckEnabled false, SetENOAutomatically false
   VAR_INPUT
      LostRetentive : Bool;   // True if retentive data are lost
      LostRTC : Bool;   // True if date and time are lost
   END_VAR
BEGIN

REGION Network 1: Braketest or mastering requred
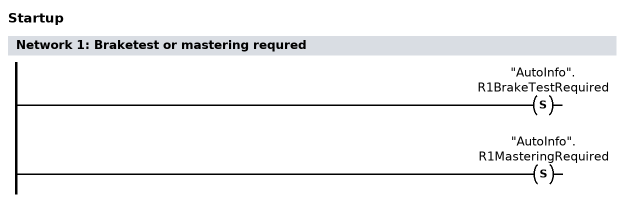
   RUNG wire#powerrail
      S_Coil( "AutoInfo".R1BrakeTestRequired )
   END_RUNG
   RUNG wire#powerrail
      S_Coil( "AutoInfo".R1MasteringRequired )
   END_RUNG
   // the same network as SCL:
   "AutoInfo".R1BrakeTestRequired := TRUE;
   "AutoInfo".R1MasteringRequired := TRUE;
END_REGION

REGION Network 2 (SCL)
       "DevicesData"."TA1-3MA".OverAcc := "StationParameters".Servo.OverAcc;
       "DevicesData"."TA1-3MA".OverDec := "StationParameters".Servo.OverDec;
       "DevicesData"."TA1-3MA".OverV := "StationParameters".Servo.OverV;
       "DevicesData"."TA1-3MA".Velocity := "StationParameters".Servo.Velocity;
END_REGION

REGION Network 3 (SCL)
   "setup_DB".minL := 100.0;
   "setup_DB".minR := "setup_DB".minL;
END_REGION
END_ORGANIZATION_BLOCK

ORGANIZATION_BLOCK "OB_IO_AccessError"   // OB122, LAD, IOAccessError
{ S7_Optimized_Access := 'TRUE' }
VERSION : 0.1
// stored: IsIECCheckEnabled false, SetENOAutomatically false
   VAR_INPUT
      BlockNr : UInt;   // Number of causing block
      Reaction : USInt;   // 0:ignore, 1:substitute, 2:skip
      Fault_ID : Byte;   // 16#42:reading, 16#43:writing
      BlockType : USInt;   // 16#01:OB, 16#02:FC, 16#03:FB, 16#04:SFC, 16#05:SFB, 16#06:DB: Type of block causing the error
      Area : USInt;   // 16#81:I, 16#82:Q: IO area where the IOaccess error occured
      DBNr : DB_ANY;   // Reserved for system
      Csg_OBNr : OB_ANY;   // Number of OB causing the error
      Csg_Prio : USInt;   // Priority of OB causing the error
      Width : USInt;   // 0:bit, 1:byte, 2:word, 3:dword, 4:lword
   END_VAR
BEGIN
END_ORGANIZATION_BLOCK

ORGANIZATION_BLOCK "OB_ProgrammingError"   // OB121, LAD, ProgrammingError
{ S7_Optimized_Access := 'TRUE' }
VERSION : 0.1
// stored: IsIECCheckEnabled false, SetENOAutomatically false
   VAR_INPUT
      BlockNr : UInt;   // Number of causing block
      Reaction : USInt;   // 0:ignore, 1:substitute, 2:skip
      Fault_ID : Byte;   // Fault identifier
      BlockType : USInt;   // 16#01:OB, 16#02:FC, 16#03:FB, 16#04:SFC, 16#05:SFB, 16#06:DB: Type of block causing the error
      Area : USInt;   // Area where the error occured
      DBNr : DB_ANY;   // DB number if Area = DB or DI
      Csg_OBNr : OB_ANY;   // Number of OB causing the error
      Csg_Prio : USInt;   // Priority of OB causing the error
      Width : USInt;   // 0:bit, 1:byte, 2:word, 3:dword, 4:lword
   END_VAR
BEGIN
END_ORGANIZATION_BLOCK

ORGANIZATION_BLOCK "OB_RackStationFailure"   // OB86, LAD, RackOrStationFailure
{ S7_Optimized_Access := 'TRUE' }
VERSION : 0.1
// stored: IsIECCheckEnabled false, SetENOAutomatically false
   VAR_INPUT
      LADDR : HW_DEVICE;   // Hardware identifier
      Event_Class : Byte;   // Event class
      Fault_ID : Byte;   // Fault identifier
   END_VAR
BEGIN
END_ORGANIZATION_BLOCK

ORGANIZATION_BLOCK "OB_Startup"   // OB100, LAD, Startup
TITLE = "Complete Restart"
{ S7_Optimized_Access := 'TRUE' }
VERSION : 0.1
// stored: AutoNumber true, IsIECCheckEnabled false, SetENOAutomatically false
   VAR_INPUT
      LostRetentive : Bool;   // True if retentive data are lost
      LostRTC : Bool;   // True if date and time are lost
   END_VAR
BEGIN
END_ORGANIZATION_BLOCK

FUNCTION_BLOCK "CylinderINC"   // FB30, LAD
{ S7_Optimized_Access := 'FALSE' }
AUTHOR : Bodorik
FAMILY : RIV
NAME : Cylinder
VERSION : 0.9
// stored: AutoNumber false, IsIECCheckEnabled false, SetENOAutomatically false, UDAEnableTagReadback false
   VAR_INPUT
      POWER_OK : Bool;
      MOVE_BASIC : Bool;
      MOVE_WORK : Bool;
      MOVE_FREE : Bool;   // QB 5
      BASIC_POSITION : Bool;   // Save cycle time
      WORK_POSITION : Bool;
      TRIGGER : Bool;
      RESET : Bool;   // QB 3
      DELAY_BASIC : Time := T#1S;
      DELAY_WORK : Time := T#1S;
      DELAY_FREE : Time := T#1S;
      ERROR_TIME : Time := T#1S;
      ValveDelay : Time;
   END_VAR
   VAR_OUTPUT
      VALVE_BASIC : Bool;   // Taking nut
      VALVE_WORK : Bool;   // 'Operate' authorization.
      CylinderStatus : "CylinderStatus";
      ERROR_BASIC : Bool;
      ERROR_WORK : Bool;
   END_VAR
   VAR_IN_OUT
      CylinderOperation : "CylinderOperation";
   END_VAR
   VAR DB_SPECIFIC
      "4l+Started" : Bool;
      InitCommandBP : Bool;
      InitCommandWP : Bool;
      BasicWorkStartWP : Bool;
      BasicWorkStartBP : Bool;
      work_valve : Bool;
      basic_valve : Bool;   // In working position
      free_valve : Bool;
      baspos_error { S7_SetPoint := 'True'} : TON_TIME;   // ton db
      workpos_error { S7_SetPoint := 'True'} : TON_TIME;
      baspos_delay { S7_SetPoint := 'True'} : TON_TIME;
      workpos_delay { S7_SetPoint := 'True'} : TON_TIME;
      CylinderOperationOld { S7_SetPoint := 'True'} : "CylinderOperation";
      IEC_Timer_0_Instance { S7_SetPoint := 'True'} : TP_TIME;
   END_VAR
   VAR
      R_TRIG_Instance { S7_SetPoint := 'True'} : R_TRIG;
   END_VAR
   VAR DB_SPECIFIC
      IEC_Timer_0_Instance_1 { S7_SetPoint := 'True'} : TP_TIME;
      IEC_Timer_0_Instance_2 { S7_SetPoint := 'True'} : TP_TIME;
      IEC_Timer_0_Instance_3 { S7_SetPoint := 'True'} : TON_TIME;
      IEC_Timer_0_Instance_4 { S7_SetPoint := 'True'} : TON_TIME;
   END_VAR
   VAR_TEMP
      et : Bool;
   END_VAR
   VAR_TEMP   // added for the SCL form of the ladder/FBD networks
      _w1 : Bool;
   END_VAR
BEGIN

REGION Network 1 (SCL): check new cylinder command
   //check if basic position req movement changed
   IF #CylinderOperation.ToBp <> #CylinderOperationOld.ToBp THEN
       #CylinderOperation.ToFp := false;
       #CylinderOperation.ToWp := false;
   END_IF;
   //check if work position req movement changed
   IF #CylinderOperation.ToWp <> #CylinderOperationOld.ToWp THEN
       #CylinderOperation.ToFp := false;
       #CylinderOperation.ToBp := false;
   END_IF;
   //check if free position req movement changed
   IF #CylinderOperation.ToFp <> #CylinderOperationOld.ToFp THEN
       #CylinderOperation.ToBp := false;
       #CylinderOperation.ToWp := false;
   END_IF;
   //store actual cylinder status to old
   #CylinderOperationOld := #CylinderOperation;
END_REGION

REGION Network 2: Start movement to basic position
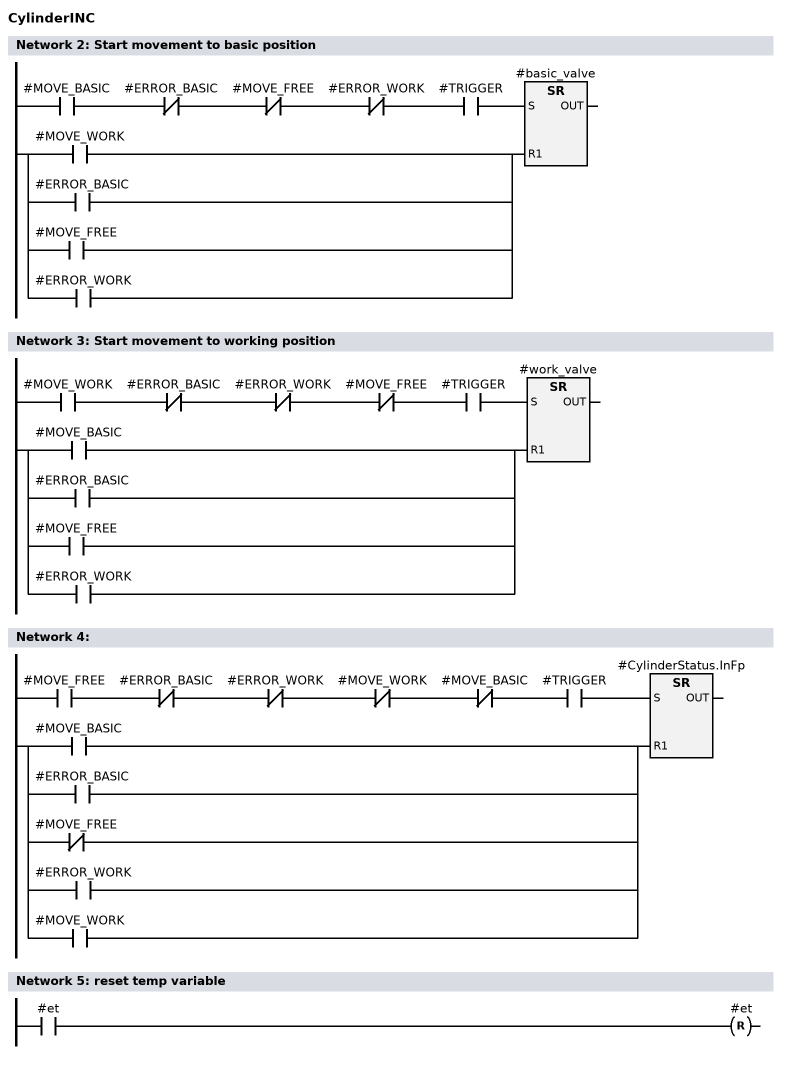
   RUNG wire#powerrail
      Contact( #MOVE_BASIC )
      I_Contact( #ERROR_BASIC )
      I_Contact( #MOVE_FREE )
      I_Contact( #ERROR_WORK )
      Contact( #TRIGGER )
      S_SR(operand := #basic_valve, r1 := wire#w1)
   END_RUNG
   RUNG wire#powerrail
      Contact( #MOVE_WORK )
   END_RUNG wire#w1
   RUNG wire#powerrail
      Contact( #ERROR_BASIC )
   END_RUNG wire#w1
   RUNG wire#powerrail
      Contact( #MOVE_FREE )
   END_RUNG wire#w1
   RUNG wire#powerrail
      Contact( #ERROR_WORK )
   END_RUNG wire#w1
   // the same network as SCL:
   IF #MOVE_BASIC AND NOT #ERROR_BASIC AND NOT #MOVE_FREE AND NOT #ERROR_WORK AND #TRIGGER THEN
       #basic_valve := TRUE;   // SR flip-flop
   END_IF;
   IF #MOVE_WORK OR #ERROR_BASIC OR #MOVE_FREE OR #ERROR_WORK THEN #basic_valve := FALSE; END_IF;
END_REGION

REGION Network 3: Start movement to working position
   RUNG wire#powerrail
      Contact( #MOVE_WORK )
      I_Contact( #ERROR_BASIC )
      I_Contact( #ERROR_WORK )
      I_Contact( #MOVE_FREE )
      Contact( #TRIGGER )
      S_SR(operand := #work_valve, r1 := wire#w1)
   END_RUNG
   RUNG wire#powerrail
      Contact( #MOVE_BASIC )
   END_RUNG wire#w1
   RUNG wire#powerrail
      Contact( #ERROR_BASIC )
   END_RUNG wire#w1
   RUNG wire#powerrail
      Contact( #MOVE_FREE )
   END_RUNG wire#w1
   RUNG wire#powerrail
      Contact( #ERROR_WORK )
   END_RUNG wire#w1
   // the same network as SCL:
   IF #MOVE_WORK AND NOT #ERROR_BASIC AND NOT #ERROR_WORK AND NOT #MOVE_FREE AND #TRIGGER THEN
       #work_valve := TRUE;   // SR flip-flop
   END_IF;
   IF #MOVE_BASIC OR #ERROR_BASIC OR #MOVE_FREE OR #ERROR_WORK THEN #work_valve := FALSE; END_IF;
END_REGION

REGION Network 4
   RUNG wire#powerrail
      Contact( #MOVE_FREE )
      I_Contact( #ERROR_BASIC )
      I_Contact( #ERROR_WORK )
      I_Contact( #MOVE_WORK )
      I_Contact( #MOVE_BASIC )
      Contact( #TRIGGER )
      S_SR(operand := #CylinderStatus.InFp, r1 := wire#w1)
   END_RUNG
   RUNG wire#powerrail
      Contact( #MOVE_BASIC )
   END_RUNG wire#w1
   RUNG wire#powerrail
      Contact( #ERROR_BASIC )
   END_RUNG wire#w1
   RUNG wire#powerrail
      I_Contact( #MOVE_FREE )
   END_RUNG wire#w1
   RUNG wire#powerrail
      Contact( #ERROR_WORK )
   END_RUNG wire#w1
   RUNG wire#powerrail
      Contact( #MOVE_WORK )
   END_RUNG wire#w1
   // the same network as SCL:
   IF #MOVE_FREE AND NOT #ERROR_BASIC AND NOT #ERROR_WORK AND NOT #MOVE_WORK AND NOT #MOVE_BASIC AND #TRIGGER THEN
       #CylinderStatus.InFp := TRUE;   // SR flip-flop
   END_IF;
   IF #MOVE_BASIC OR #ERROR_BASIC OR NOT #MOVE_FREE OR #ERROR_WORK OR #MOVE_WORK THEN
       #CylinderStatus.InFp := FALSE;
   END_IF;
END_REGION

REGION Network 5: reset temp variable
   RUNG wire#powerrail
      Contact( #et )
      R_Coil( #et )
   END_RUNG
   // the same network as SCL:
   IF #et THEN #et := FALSE; END_IF;
END_REGION

REGION Network 6 (FBD): Error movement to basic position
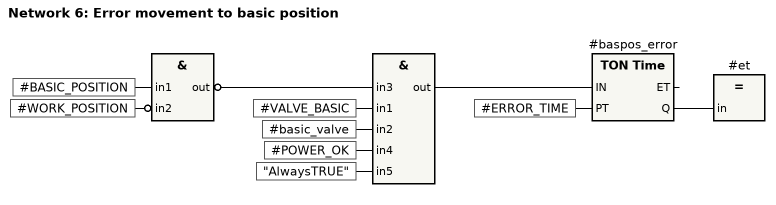
   #baspos_error(IN := NOT (#BASIC_POSITION AND NOT #WORK_POSITION) AND #VALVE_BASIC AND #basic_valve AND #POWER_OK AND "AlwaysTRUE",   // TON
                 PT := #ERROR_TIME);
   #et := #baspos_error.Q;
END_REGION

REGION Network 7: Set basic position error
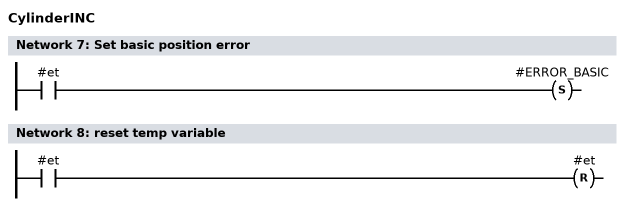
   RUNG wire#powerrail
      Contact( #et )
      S_Coil( #ERROR_BASIC )
   END_RUNG
   // the same network as SCL:
   IF #et THEN #ERROR_BASIC := TRUE; END_IF;
END_REGION

REGION Network 8: reset temp variable
   RUNG wire#powerrail
      Contact( #et )
      R_Coil( #et )
   END_RUNG
   // the same network as SCL:
   IF #et THEN #et := FALSE; END_IF;
END_REGION

REGION Network 9 (FBD): Error movement to working position
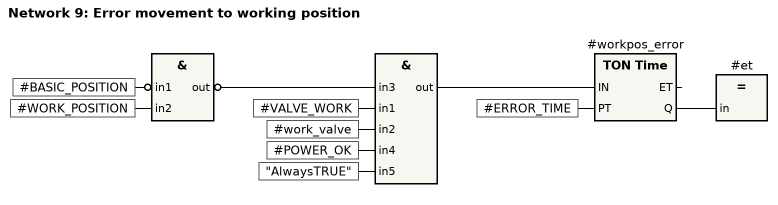
   #workpos_error(IN := NOT (NOT #BASIC_POSITION AND #WORK_POSITION) AND #VALVE_WORK AND #work_valve AND #POWER_OK AND "AlwaysTRUE",   // TON
                  PT := #ERROR_TIME);
   #et := #workpos_error.Q;
END_REGION

REGION Network 10: Set working position error
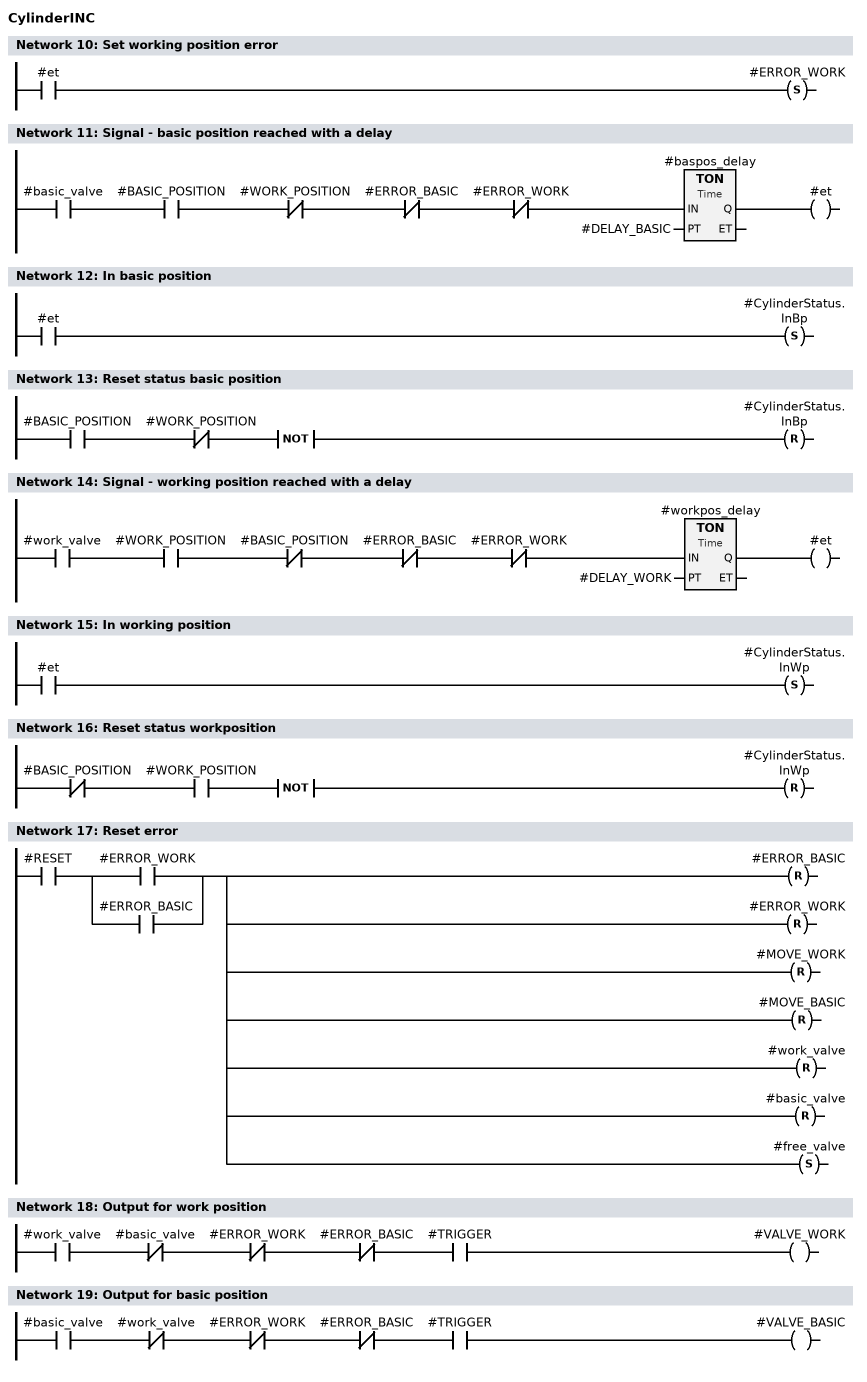
   RUNG wire#powerrail
      Contact( #et )
      S_Coil( #ERROR_WORK )
   END_RUNG
   // the same network as SCL:
   IF #et THEN #ERROR_WORK := TRUE; END_IF;
END_REGION

REGION Network 11: Signal - basic position reached with a delay
   RUNG wire#powerrail
      Contact( #basic_valve )
      Contact( #BASIC_POSITION )
      I_Contact( #WORK_POSITION )
      I_Contact( #ERROR_BASIC )
      I_Contact( #ERROR_WORK )
      { S7_Templates := "time_type := Time" } #baspos_delay.TON(pt := #DELAY_BASIC, et =>)
      Coil( #et )
   END_RUNG
   // the same network as SCL:
   #baspos_delay(PT := #DELAY_BASIC,   // TON
                 IN := #basic_valve AND #BASIC_POSITION AND NOT #WORK_POSITION AND NOT #ERROR_BASIC AND NOT #ERROR_WORK);
   #et := #baspos_delay.Q;
END_REGION

REGION Network 12: In basic position
   RUNG wire#powerrail
      Contact( #et )
      S_Coil( #CylinderStatus.InBp )
   END_RUNG
   // the same network as SCL:
   IF #et THEN #CylinderStatus.InBp := TRUE; END_IF;
END_REGION

REGION Network 13: Reset status basic position
   RUNG wire#powerrail
      Contact( #BASIC_POSITION )
      I_Contact( #WORK_POSITION )
      Not()
      R_Coil( #CylinderStatus.InBp )
   END_RUNG
   // the same network as SCL:
   IF NOT (#BASIC_POSITION AND NOT #WORK_POSITION) THEN #CylinderStatus.InBp := FALSE; END_IF;
END_REGION

REGION Network 14: Signal - working position reached with a delay
   RUNG wire#powerrail
      Contact( #work_valve )
      Contact( #WORK_POSITION )
      I_Contact( #BASIC_POSITION )
      I_Contact( #ERROR_BASIC )
      I_Contact( #ERROR_WORK )
      { S7_Templates := "time_type := Time" } #workpos_delay.TON(pt := #DELAY_WORK, et =>)
      Coil( #et )
   END_RUNG
   // the same network as SCL:
   #workpos_delay(PT := #DELAY_WORK,   // TON
                  IN := #work_valve AND #WORK_POSITION AND NOT #BASIC_POSITION AND NOT #ERROR_BASIC AND NOT #ERROR_WORK);
   #et := #workpos_delay.Q;
END_REGION

REGION Network 15: In working position
   RUNG wire#powerrail
      Contact( #et )
      S_Coil( #CylinderStatus.InWp )
   END_RUNG
   // the same network as SCL:
   IF #et THEN #CylinderStatus.InWp := TRUE; END_IF;
END_REGION

REGION Network 16: Reset status workposition
   RUNG wire#powerrail
      I_Contact( #BASIC_POSITION )
      Contact( #WORK_POSITION )
      Not()
      R_Coil( #CylinderStatus.InWp )
   END_RUNG
   // the same network as SCL:
   IF NOT (NOT #BASIC_POSITION AND #WORK_POSITION) THEN #CylinderStatus.InWp := FALSE; END_IF;
END_REGION

REGION Network 17: Reset error
   RUNG wire#powerrail
      Contact( #RESET )
      wire#w1
      Contact( #ERROR_WORK )
      wire#w2
      R_Coil( #ERROR_BASIC )
   END_RUNG
   RUNG wire#w1
      Contact( #ERROR_BASIC )
   END_RUNG wire#w2
   RUNG wire#w2
      R_Coil( #ERROR_WORK )
   END_RUNG
   RUNG wire#w2
      R_Coil( #MOVE_WORK )
   END_RUNG
   RUNG wire#w2
      R_Coil( #MOVE_BASIC )
   END_RUNG
   RUNG wire#w2
      R_Coil( #work_valve )
   END_RUNG
   RUNG wire#w2
      R_Coil( #basic_valve )
   END_RUNG
   RUNG wire#w2
      S_Coil( #free_valve )
   END_RUNG
   // the same network as SCL:
   #_w1 := #RESET AND (#ERROR_WORK OR #ERROR_BASIC);
   IF #_w1 THEN
       #ERROR_BASIC := FALSE;
       #ERROR_WORK := FALSE;
       #MOVE_WORK := FALSE;
       #MOVE_BASIC := FALSE;
       #work_valve := FALSE;
       #basic_valve := FALSE;
       #free_valve := TRUE;
   END_IF;
END_REGION

REGION Network 18: Output for work position
   RUNG wire#powerrail
      Contact( #work_valve )
      I_Contact( #basic_valve )
      I_Contact( #ERROR_WORK )
      I_Contact( #ERROR_BASIC )
      Contact( #TRIGGER )
      Coil( #VALVE_WORK )
   END_RUNG
   // the same network as SCL:
   #VALVE_WORK := #work_valve AND NOT #basic_valve AND NOT #ERROR_WORK AND NOT #ERROR_BASIC AND #TRIGGER;
END_REGION

REGION Network 19: Output for basic position
   RUNG wire#powerrail
      Contact( #basic_valve )
      I_Contact( #work_valve )
      I_Contact( #ERROR_WORK )
      I_Contact( #ERROR_BASIC )
      Contact( #TRIGGER )
      Coil( #VALVE_BASIC )
   END_RUNG
   // the same network as SCL:
   #VALVE_BASIC := #basic_valve AND NOT #work_valve AND NOT #ERROR_WORK AND NOT #ERROR_BASIC AND #TRIGGER;
END_REGION

REGION Network 20 (SCL)
   #R_TRIG_Instance(CLK:=#POWER_OK
   );

   IF #R_TRIG_Instance.Q THEN
       #"4l+Started" := TRUE;

   END_IF;

   IF #MOVE_BASIC AND #"4l+Started" THEN

       #InitCommandBP := true;
   END_IF;
   IF #MOVE_WORK AND #"4l+Started" THEN

       #InitCommandWP := true;
   END_IF;

   #IEC_Timer_0_Instance_1(IN:=#InitCommandBP,
                               PT:=t#10ms,
                               Q=>#BasicWorkStartBP
       );
   #IEC_Timer_0_Instance_2(IN:=#InitCommandWP,
                               PT:=t#10ms,
                               Q=>#BasicWorkStartWP
   );


   IF #BasicWorkStartBP  THEN
       #VALVE_WORK := TRUE;
       #VALVE_BASIC := FALSE;
       ;

   END_IF;

   IF #BasicWorkStartWP THEN
       #VALVE_WORK := FALSE;
       #VALVE_BASIC := TRUE;
       ;

   END_IF;

   IF NOT #IEC_Timer_0_Instance_1.Q AND #InitCommandBP THEN
       #VALVE_WORK := FALSE;
       #VALVE_BASIC := TRUE;
       #"4l+Started" := FALSE;
       #InitCommandBP := FALSE;
       ;
   END_IF;
   IF NOT #IEC_Timer_0_Instance_2.Q AND #InitCommandWP THEN
       #VALVE_WORK := TRUE;
       #VALVE_BASIC := FALSE;
       #"4l+Started" := FALSE;
       #InitCommandWP := FALSE;
       ;
   END_IF;
END_REGION
END_FUNCTION_BLOCK

FUNCTION "FC_ByteToCharacters" : Void   // FC1071, LAD
{ S7_Optimized_Access := 'FALSE' }
VERSION : 0.1
// stored: AutoNumber false, IsIECCheckEnabled false, SetENOAutomatically false, UDAEnableTagReadback false
   VAR_INPUT
      iByte : Byte;
   END_VAR
   VAR_OUTPUT
      qChar1 : Char;
      qChar2 : Char;
   END_VAR
   VAR_TEMP
      "b" : Byte;
      char1_value : UInt;
      char2_value : UInt;
   END_VAR
   VAR_TEMP   // added for the SCL form of the ladder/FBD networks
      _w1 : Bool;
      _w2 : Bool;
   END_VAR
BEGIN

REGION Network 1: Load input byte to temporary
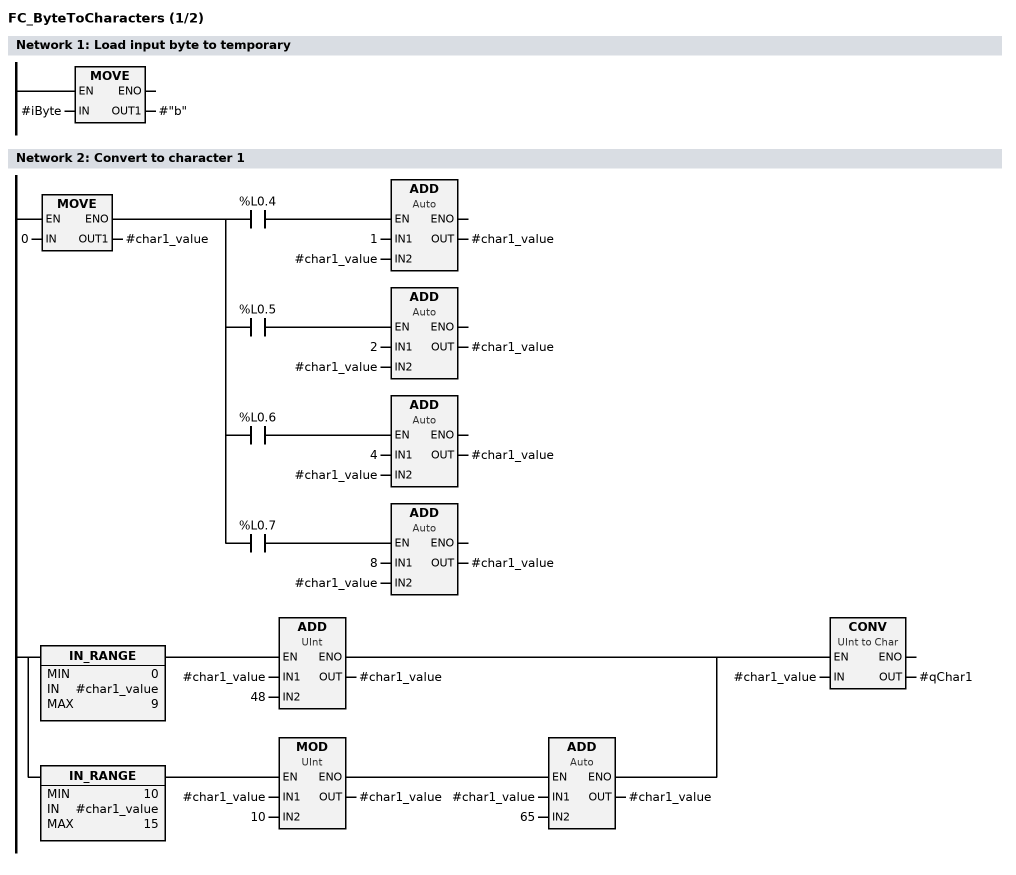
   RUNG wire#powerrail
      Move(in := #iByte, out1 => #"b")
   END_RUNG
   // the same network as SCL:
   #"b" := #iByte;
END_REGION

REGION Network 2: Convert to character 1
   RUNG wire#powerrail
      Move(in := 0, out1 => #char1_value)
      wire#w1
      Contact( %L0.4 )
      Add(in1 := 1, in2 := #char1_value, out => #char1_value)
   END_RUNG
   RUNG wire#w1
      Contact( %L0.5 )
      Add(in1 := 2, in2 := #char1_value, out => #char1_value)
   END_RUNG
   RUNG wire#w1
      Contact( %L0.6 )
      Add(in1 := 4, in2 := #char1_value, out => #char1_value)
   END_RUNG
   RUNG wire#w1
      Contact( %L0.7 )
      Add(in1 := 8, in2 := #char1_value, out => #char1_value)
   END_RUNG
   RUNG wire#powerrail
      { S7_Templates := "SrcType := UInt" } InRange(min := 0, in := #char1_value, max := 9)
      { S7_Templates := "SrcType := UInt" } Add(in1 := #char1_value, in2 := 48, out => #char1_value)
      wire#w2
      { S7_Templates := "[SrcType := UInt, DestType := Char]" } Convert(in := #char1_value, out => #qChar1)
   END_RUNG
   RUNG wire#powerrail
      { S7_Templates := "SrcType := UInt" } InRange(min := 10, in := #char1_value, max := 15)
      { S7_Templates := "SrcType := UInt" } Mod(in1 := #char1_value, in2 := 10, out => #char1_value)
      Add(in1 := #char1_value, in2 := 65, out => #char1_value)
   END_RUNG wire#w2
   // the same network as SCL:
   #char1_value := 0;
   IF %L0.4 THEN #char1_value := 1 + #char1_value; END_IF;
   IF %L0.5 THEN #char1_value := 2 + #char1_value; END_IF;
   IF %L0.6 THEN #char1_value := 4 + #char1_value; END_IF;
   IF %L0.7 THEN #char1_value := 8 + #char1_value; END_IF;
   #_w1 := (0 <= #char1_value) AND (#char1_value <= 9);
   IF #_w1 THEN #char1_value := #char1_value + 48; END_IF;
   #_w2 := (10 <= #char1_value) AND (#char1_value <= 15);
   IF #_w2 THEN
       #char1_value := #char1_value MOD 10;
       #char1_value := #char1_value + 65;
   END_IF;
   IF #_w1 OR #_w2 THEN #qChar1 := UINT_TO_CHAR(#char1_value); END_IF;
END_REGION

REGION Network 3: Convert to character 2
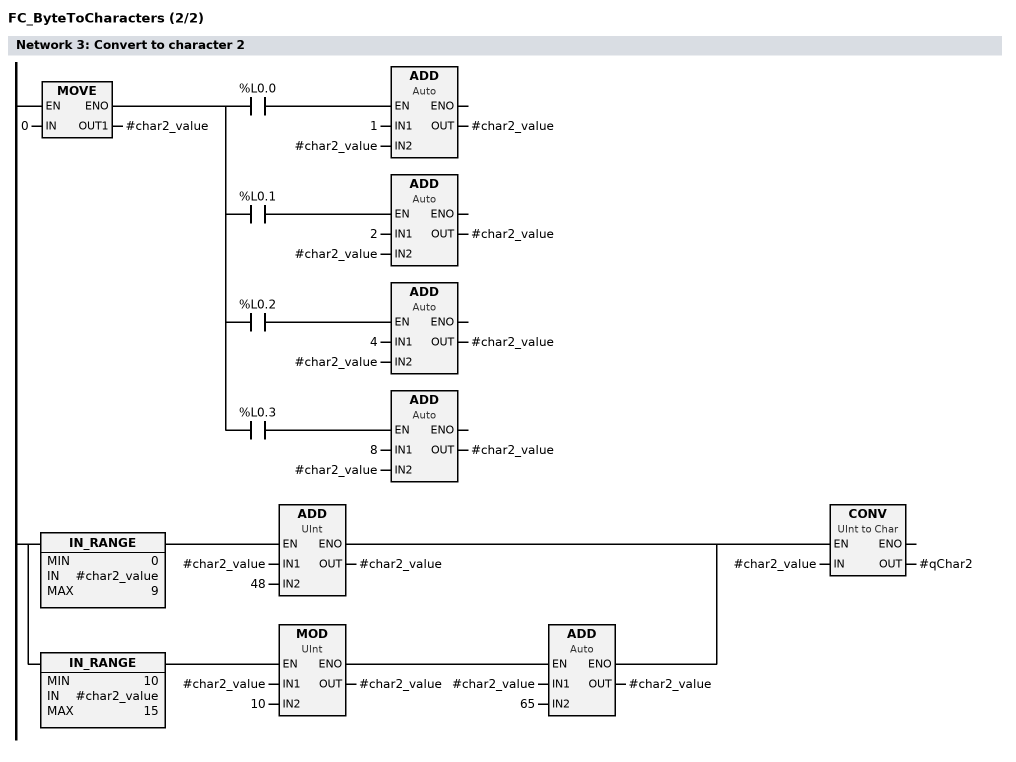
   RUNG wire#powerrail
      Move(in := 0, out1 => #char2_value)
      wire#w1
      Contact( %L0.0 )
      Add(in1 := 1, in2 := #char2_value, out => #char2_value)
   END_RUNG
   RUNG wire#w1
      Contact( %L0.1 )
      Add(in1 := 2, in2 := #char2_value, out => #char2_value)
   END_RUNG
   RUNG wire#w1
      Contact( %L0.2 )
      Add(in1 := 4, in2 := #char2_value, out => #char2_value)
   END_RUNG
   RUNG wire#w1
      Contact( %L0.3 )
      Add(in1 := 8, in2 := #char2_value, out => #char2_value)
   END_RUNG
   RUNG wire#powerrail
      { S7_Templates := "SrcType := UInt" } InRange(min := 0, in := #char2_value, max := 9)
      { S7_Templates := "SrcType := UInt" } Add(in1 := #char2_value, in2 := 48, out => #char2_value)
      wire#w2
      { S7_Templates := "[SrcType := UInt, DestType := Char]" } Convert(in := #char2_value, out => #qChar2)
   END_RUNG
   RUNG wire#powerrail
      { S7_Templates := "SrcType := UInt" } InRange(min := 10, in := #char2_value, max := 15)
      { S7_Templates := "SrcType := UInt" } Mod(in1 := #char2_value, in2 := 10, out => #char2_value)
      Add(in1 := #char2_value, in2 := 65, out => #char2_value)
   END_RUNG wire#w2
   // the same network as SCL:
   #char2_value := 0;
   IF %L0.0 THEN #char2_value := 1 + #char2_value; END_IF;
   IF %L0.1 THEN #char2_value := 2 + #char2_value; END_IF;
   IF %L0.2 THEN #char2_value := 4 + #char2_value; END_IF;
   IF %L0.3 THEN #char2_value := 8 + #char2_value; END_IF;
   #_w1 := (0 <= #char2_value) AND (#char2_value <= 9);
   IF #_w1 THEN #char2_value := #char2_value + 48; END_IF;
   #_w2 := (10 <= #char2_value) AND (#char2_value <= 15);
   IF #_w2 THEN
       #char2_value := #char2_value MOD 10;
       #char2_value := #char2_value + 65;
   END_IF;
   IF #_w1 OR #_w2 THEN #qChar2 := UINT_TO_CHAR(#char2_value); END_IF;
END_REGION
END_FUNCTION

FUNCTION_BLOCK "1. DMC_setConnection"   // FB2001, LAD
{ S7_Optimized_Access := 'FALSE' }
AUTHOR : bartz
VERSION : 0.1
// stored: AutoNumber false, IsIECCheckEnabled false, SetENOAutomatically false, UDAEnableTagReadback false
   VAR DB_SPECIFIC
      Connection : Struct
         IPAddress : WString := WSTRING#'';   // IP without the opc.tcp:// / Server IP Address (e.g. 10.223.41.34)
         ServerPort : WString := WSTRING#'';   // Only numbers / Server port (e.g. 58710/PCoUaServer)
         PlantID : WString := WSTRING#'';   // Unique plant id defined by GIS (e.g. P1, P2)
         PLC_ID : WString := WSTRING#'';   // Unique plc id defined by GIS
         OperationMode : Bool := False;   // Operation mode: test or production
      END_STRUCT;
      Controllers : Struct
         opcUaConnect : Bool;
         opcUaMethodCall : Bool;
         opcUaMethodIndex : SInt;
         opcUaConnected { S7_SetPoint := 'True'} : Bool;
         opcUaDone : Bool;
         opcUaBusy : Bool;
         opcUaError : Bool;
         opcUaStatus : Word;
         opcUaDiagnostics : "typeFbDiagnostics";
      END_STRUCT;
      Auxiliar : Struct   // Method fb's call auxiliar variables
         endpointTemp : String[254];
         idx : Int;
         timeout : Bool;
         life : Bool;
         closedRequested : Bool;
         tryAgain : Bool;
         attempts : Int;
      END_STRUCT;
      Timers : Struct
         timeoutCallMethod : TON_TIME;
         forceReconnection { S7_SetPoint := 'True'} : TON_TIME;
         tryAgain { S7_SetPoint := 'True'} : TON_TIME;
      END_STRUCT;
      CallBuffer : Array[0..#nMethods] of Bool;
   END_VAR
   VAR_TEMP
      methodInputs : Variant;
      methodOutputs : Variant;
      retVal : Int;
   END_VAR
   VAR CONSTANT
      nMethods : Int := 9;
      callTimeout : Time := T#5s;
      nAttempts : Int := 2;
   END_VAR
BEGIN

REGION Network 1 (SCL): Set connection
   // Assign data from MII_PARAMETERS [DB2020]
   #Connection.IPAddress := "MII_Parameters".Connection.IPAddress;
   #Connection.ServerPort := "MII_Parameters".Connection.ServerPort;
   #Connection.PlantID := "MII_Parameters".Connection.PlantID;
   #Connection.PLC_ID := "MII_Parameters".Connection.PLC_ID;
   #Connection.OperationMode := "MII_Parameters".Connection.OperationMode;

   // Configure IP + Port to establish connection
   IF "MII_Interface_Configuration".Connection.ServerEndpointUrl <> #Auxiliar.endpointTemp OR #Connection.IPAddress = WSTRING#'' OR #Connection.ServerPort = WSTRING#'' THEN
       #Controllers.opcUaConnect := FALSE;
       #Auxiliar.endpointTemp := "MII_Interface_Configuration".Connection.ServerEndpointUrl;
   ELSE
       "MII_Interface_Configuration".Connection.ServerEndpointUrl := WSTRING_TO_STRING(CONCAT_WSTRING(IN1 := WSTRING#'opc.tcp://', IN2 := #Connection.IPAddress, IN3 := WSTRING#':', IN4 := #Connection.ServerPort, IN5 := WSTRING#'/PCoUaServer'));

   END_IF;

   // Manual reconnection
   IF NOT #Auxiliar.life AND "MII_Parameters".Commands.forceReconnection THEN
       #Controllers.opcUaConnect := TRUE;
       IF "0. OpcUaClient_DB".statOpcUaRequests.disconnect THEN
           // Reset disconnect button 
           "0. OpcUaClient_DB".statOpcUaRequests.disconnect := FALSE;
       END_IF;
   END_IF;

   //Force reconnection timer
   #Timers.forceReconnection(IN := "MII_Parameters".Commands.forceReconnection,
                             PT := t#10s,
                             Q => #Auxiliar.life);

   // Reset force reconnection after 10s
   IF #Auxiliar.life THEN
       "MII_Parameters".Commands.forceReconnection := FALSE;
   END_IF;

   //Method call timeout
   #Timers.timeoutCallMethod(IN := #Controllers.opcUaMethodCall,
                             PT := t#10s,
                             Q => #Auxiliar.timeout);
END_REGION

REGION Network 2 (SCL): Prepare method call
   //Open connection if method called on buffer
   FOR #Auxiliar.idx := 0 TO #nMethods DO
       IF #Controllers.opcUaMethodCall = FALSE AND #CallBuffer[#Auxiliar.idx] = TRUE AND NOT #Auxiliar.closedRequested THEN
           #Controllers.opcUaConnect := TRUE;
       END_IF;
   END_FOR;

   IF NOT #Controllers.opcUaConnected AND #Auxiliar.closedRequested THEN
       #Auxiliar.closedRequested := False;
   END_IF;




   IF #Controllers.opcUaConnected = FALSE OR #Auxiliar.closedRequested THEN
       //DOWNGRADED MODE
       #Controllers.opcUaMethodCall := FALSE;

   ELSE
       //NORMAL MODE
       FOR #Auxiliar.idx := 0 TO #nMethods DO
           IF #Controllers.opcUaMethodCall = FALSE AND #CallBuffer[#Auxiliar.idx] = TRUE THEN
               #Controllers.opcUaMethodIndex := INT_TO_SINT(#Auxiliar.idx);
               #Controllers.opcUaMethodCall := TRUE;
           END_IF;
       END_FOR;

       REGION SWITCH CASE
           CASE #Controllers.opcUaMethodIndex OF
               0:  //M000_PRODUCTION_DECLARATION
                   #methodInputs := REF("MII_Interface_Data".MII_METHODS."M000_PRODUCTION_DECLARATION".Inputs);
                   VariantPut(SRC := "MII_Interface_Data".MII_METHODS."M000_PRODUCTION_DECLARATION".Inputs,
                              DST := #methodInputs);
                   #methodOutputs := REF("MII_Interface_Data".MII_METHODS."M000_PRODUCTION_DECLARATION".Outputs);
                   VariantPut(SRC := "MII_Interface_Data".MII_METHODS."M000_PRODUCTION_DECLARATION".Outputs,
                              DST := #methodOutputs);

               1:  //M001_GET_LOCAL_TIME
                   #methodOutputs := REF("MII_Interface_Data".MII_METHODS."M001_GET_LOCAL_TIME".Outputs);
                   VariantPut(SRC := "MII_Interface_Data".MII_METHODS."M001_GET_LOCAL_TIME".Outputs,
                              DST := #methodOutputs);

               2:  //M101_SCRAP_DECLARATION
                   #methodInputs := REF("MII_Interface_Data".MII_METHODS."M101_SCRAP_DECLARATION".Inputs);
                   VariantPut(SRC := "MII_Interface_Data".MII_METHODS."M101_SCRAP_DECLARATION".Inputs,
                              DST := #methodInputs);
                   #methodOutputs := REF("MII_Interface_Data".MII_METHODS."M101_SCRAP_DECLARATION".Outputs);
                   VariantPut(SRC := "MII_Interface_Data".MII_METHODS."M101_SCRAP_DECLARATION".Outputs,
                              DST := #methodOutputs);

               3:  //M003_GENERATE_ALERT
                   #methodInputs := REF("MII_Interface_Data".MII_METHODS."M003_GENERATE_ALERT".Inputs);
                   VariantPut(SRC := "MII_Interface_Data".MII_METHODS."M003_GENERATE_ALERT".Inputs,
                              DST := #methodInputs);
                   #methodOutputs := REF("MII_Interface_Data".MII_METHODS."M003_GENERATE_ALERT".Outputs);
                   VariantPut(SRC := "MII_Interface_Data".MII_METHODS."M003_GENERATE_ALERT".Outputs,
                              DST := #methodOutputs);

               4:  //M102_REWORK_DECLARATION
                   #methodInputs := REF("MII_Interface_Data".MII_METHODS."M102_REWORK_DECLARATION".Inputs);
                   VariantPut(SRC := "MII_Interface_Data".MII_METHODS."M102_REWORK_DECLARATION".Inputs,
                              DST := #methodInputs);
                   #methodOutputs := REF("MII_Interface_Data".MII_METHODS."M102_REWORK_DECLARATION".Outputs);
                   VariantPut(SRC := "MII_Interface_Data".MII_METHODS."M102_REWORK_DECLARATION".Outputs,
                              DST := #methodOutputs);

               5:  //M002_GET_PLANTS
                   #methodOutputs := REF("MII_Interface_Data".MII_METHODS."M002_GET_PLANTS".Outputs);
                   VariantPut(SRC := "MII_Interface_Data".MII_METHODS.M002_GET_PLANTS.Outputs,
                              DST := #methodOutputs);

               6: //NON TRS
                   #methodInputs := REF("MII_Interface_Data".MII_METHODS.M004_NTRS.Inputs);
                   VariantPut(SRC := "MII_Interface_Data".MII_METHODS.M004_NTRS.Inputs,
                              DST := #methodInputs);
                   #methodOutputs := REF("MII_Interface_Data".MII_METHODS.M004_NTRS.Outputs);
                   VariantPut(SRC := "MII_Interface_Data".MII_METHODS.M004_NTRS.Outputs,
                              DST := #methodOutputs);

               7: //PY
                   #methodInputs := REF("MII_Interface_Data".MII_METHODS.M103_PY.Inputs);
                   VariantPut(SRC := "MII_Interface_Data".MII_METHODS.M103_PY.Inputs,
                              DST := #methodInputs);
                   #methodOutputs := REF("MII_Interface_Data".MII_METHODS.M103_PY.Outputs);
                   VariantPut(SRC := "MII_Interface_Data".MII_METHODS.M103_PY.Outputs,
                              DST := #methodOutputs);

               8: //VARABILITY
                   #methodInputs := REF("MII_Interface_Data".MII_METHODS.M005_VARIABILITY.Inputs);
                   VariantPut(SRC := "MII_Interface_Data".MII_METHODS.M005_VARIABILITY.Inputs,
                              DST := #methodInputs);
                   #methodOutputs := REF("MII_Interface_Data".MII_METHODS.M005_VARIABILITY.Outputs);
                   VariantPut(SRC := "MII_Interface_Data".MII_METHODS.M005_VARIABILITY.Outputs,
                              DST := #methodOutputs);

           END_CASE;
       END_REGION ;
   END_IF;
END_REGION

REGION Network 3: Call client fb
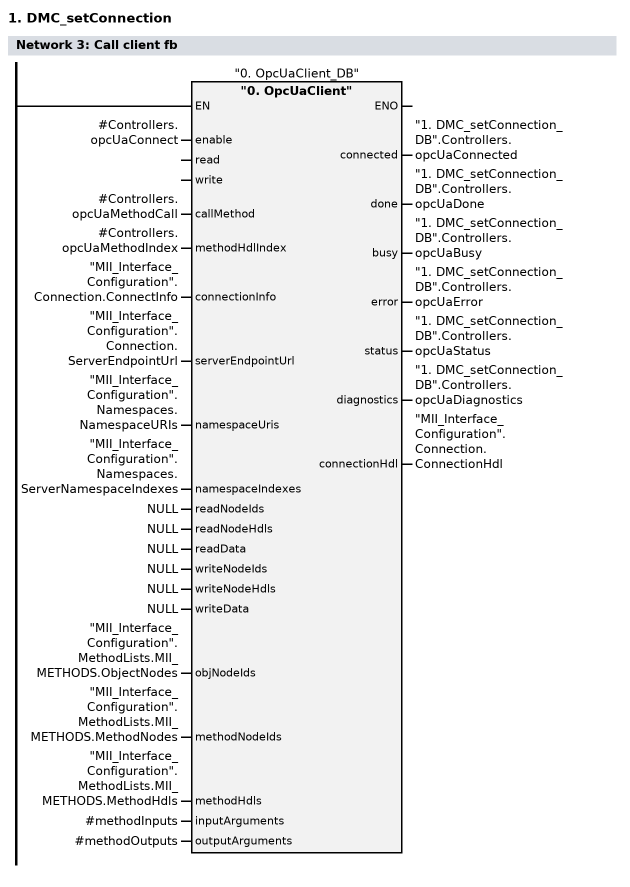
   RUNG wire#powerrail
      "0. OpcUaClient_DB"(enable := #Controllers.opcUaConnect, read :=, write :=, callMethod := #Controllers.opcUaMethodCall, methodHdlIndex := #Controllers.opcUaMethodIndex, connectionInfo := "MII_Interface_Configuration".Connection.ConnectInfo, serverEndpointUrl := "MII_Interface_Configuration".Connection.ServerEndpointUrl, namespaceUris := "MII_Interface_Configuration".Namespaces.NamespaceURIs, namespaceIndexes := "MII_Interface_Configuration".Namespaces.ServerNamespaceIndexes, readNodeIds := NULL, readNodeHdls := NULL, readData := NULL, writeNodeIds := NULL, writeNodeHdls := NULL, writeData := NULL, objNodeIds := "MII_Interface_Configuration".MethodLists.MII_METHODS.ObjectNodes, methodNodeIds := "MII_Interface_Configuration".MethodLists.MII_METHODS.MethodNodes, methodHdls := "MII_Interface_Configuration".MethodLists.MII_METHODS.MethodHdls, inputArguments := #methodInputs, outputArguments := #methodOutputs, connected => "1. DMC_setConnection_DB".Controllers.opcUaConnected, done => "1. DMC_setConnection_DB".Controllers.opcUaDone, busy => "1. DMC_setConnection_DB".Controllers.opcUaBusy, error => "1. DMC_setConnection_DB".Controllers.opcUaError, status => "1. DMC_setConnection_DB".Controllers.opcUaStatus, diagnostics => "1. DMC_setConnection_DB".Controllers.opcUaDiagnostics, connectionHdl => "MII_Interface_Configuration".Connection.ConnectionHdl)
   END_RUNG
   // the same network as SCL:
   "0. OpcUaClient_DB"(enable := #Controllers.opcUaConnect,   // "0. OpcUaClient"
                       callMethod := #Controllers.opcUaMethodCall,
                       methodHdlIndex := #Controllers.opcUaMethodIndex,
                       connectionInfo := "MII_Interface_Configuration".Connection.ConnectInfo,
                       serverEndpointUrl := "MII_Interface_Configuration".Connection.ServerEndpointUrl,
                       namespaceUris := "MII_Interface_Configuration".Namespaces.NamespaceURIs,
                       namespaceIndexes := "MII_Interface_Configuration".Namespaces.ServerNamespaceIndexes,
                       readNodeIds := NULL,
                       readNodeHdls := NULL,
                       readData := NULL,
                       writeNodeIds := NULL,
                       writeNodeHdls := NULL,
                       writeData := NULL,
                       objNodeIds := "MII_Interface_Configuration".MethodLists.MII_METHODS.ObjectNodes,
                       methodNodeIds := "MII_Interface_Configuration".MethodLists.MII_METHODS.MethodNodes,
                       methodHdls := "MII_Interface_Configuration".MethodLists.MII_METHODS.MethodHdls,
                       inputArguments := #methodInputs,
                       outputArguments := #methodOutputs,
                       connected => "1. DMC_setConnection_DB".Controllers.opcUaConnected,
                       done => "1. DMC_setConnection_DB".Controllers.opcUaDone,
                       busy => "1. DMC_setConnection_DB".Controllers.opcUaBusy,
                       error => "1. DMC_setConnection_DB".Controllers.opcUaError,
                       status => "1. DMC_setConnection_DB".Controllers.opcUaStatus,
                       diagnostics => "1. DMC_setConnection_DB".Controllers.opcUaDiagnostics,
                       connectionHdl => "MII_Interface_Configuration".Connection.ConnectionHdl);
END_REGION

REGION Network 4 (SCL): Post method call
   IF #Controllers.opcUaMethodCall AND (#Controllers.opcUaDone OR #Auxiliar.timeout OR #Controllers.opcUaError) THEN
       REGION SWITCH CASE
           CASE #Controllers.opcUaMethodIndex OF
               0:  //M000_PRODUCTION_DECLARATION
                   //Send the inputs and the output to the HMI
                   "MII_Parameters".M000_Status.Inputs := "MII_Interface_Data".MII_METHODS.M000_PRODUCTION_DECLARATION.Inputs;
                   "MII_Parameters".M000_Status.Outputs := "MII_Interface_Data".MII_METHODS.M000_PRODUCTION_DECLARATION.Outputs;


                   IF "MII_Interface_Data".MII_METHODS.M000_PRODUCTION_DECLARATION.Outputs.SUCCESS_FLAG = 0 OR #Auxiliar.timeout THEN
                       //Write error status
                       IF #Auxiliar.timeout THEN
                           "MII_Parameters".M000_Status.status := Wstring#'TimeoutERROR';
                       ELSE
                           "MII_Parameters".M000_Status.status := "MII_Interface_Data".MII_METHODS.M000_PRODUCTION_DECLARATION.Outputs.STATUS_MESSAGE;
                       END_IF;

                       //Get error timestamp 
                       #retVal := RD_LOC_T("MII_Parameters".M000_Status.timestamp);

                       //Set error trigger to HMI store values
                       //Note: HMI must reset this tag after writing the file
                       "MII_Parameters".M000_Status.error := TRUE;
                   ELSE
                       //Reset error if declaration is ok
                       "MII_Parameters".M000_Status.error := FALSE;
                       "MII_Parameters".M000_Status.status := "MII_Interface_Data".MII_METHODS.M000_PRODUCTION_DECLARATION.Outputs.STATUS_MESSAGE;
                   END_IF;

                   //Reset test command and add one to the auxiliar cycle counter
                   IF "MII_Parameters".Commands.testProdDeclaration THEN
                       "MII_Parameters".Commands.testProdDeclaration := FALSE;
                       "MII_Parameters".Commands.auxTestProdDeclaration := "MII_Parameters".Commands.auxTestProdDeclaration + 1;
                   END_IF;

               1: //M002_GET_LOCAL_TIME
                   IF #Auxiliar.timeout THEN
                       "MII_Parameters".M002_Status.status := WSTRING#'TimeoutERROR';
                   ELSE
                       //Overwrite system time
                       #retVal := WR_LOC_T(LOCTIME := "MII_Interface_Data".MII_METHODS.M001_GET_LOCAL_TIME.Outputs.DATETIME_LOCAL, DST := TRUE);

                       //Set M002_status
                       "MII_Parameters".M002_Status.localTime := "MII_Interface_Data".MII_METHODS.M001_GET_LOCAL_TIME.Outputs.DATETIME_LOCAL;
                       "MII_Parameters".M002_Status.status := WSTRING#'OK';

                       //Reset command after calling the method
                       "MII_Parameters".Commands.getLocalTime := FALSE;
                   END_IF;

               2: //TO BE DEVELOPED
                   ;

               3: //TO BE DEVELOPED
                   ;

               4: //TO BE DEVELOPED
                   ;

               5: //TO BE DEVELOPED
                   ;

               6: //TO BE DEVELOPED
                   ;

               7: //TO BE DEVELOPED
                   ;

               8: //TO BE DEVELOPED
                   ;

           END_CASE;
       END_REGION

       IF #Auxiliar.attempts <= #nAttempts AND #CallBuffer[0] AND (#Controllers.opcUaError OR #Auxiliar.timeout) THEN
           #Auxiliar.attempts := #Auxiliar.attempts + 1;
           #Auxiliar.closedRequested := true;
           #Controllers.opcUaConnect := False;

       ELSE
           //RESET METHOD INDEX
           #CallBuffer[#Controllers.opcUaMethodIndex] := FALSE;
           #Auxiliar.attempts := 0;
           //Close #Connection IF no called method on buffer
           #Auxiliar.closedRequested := true;
           FOR #Auxiliar.idx := 0 TO #nMethods DO
               IF #CallBuffer[#Auxiliar.idx] = true THEN
                   #Auxiliar.closedRequested := false;
               END_IF;
           END_FOR;
           IF #Auxiliar.closedRequested THEN
               #Controllers.opcUaConnect := False;
               #Auxiliar.closedRequested := False;
           END_IF;
       END_IF;

       //RESET METHOD TAG
       #Controllers.opcUaMethodCall := FALSE;
   END_IF;
END_REGION

REGION Network 5 (SCL): Device diagnostics
   // Read diagnostic status
   "MII_Parameters".Connection_Status.opcUaConnected := #Controllers.opcUaConnected;
   "MII_Parameters".Connection_Status.opcUaError := #Controllers.opcUaError;
   "MII_Parameters".Connection_Status.opcUaStatus := #Controllers.opcUaStatus;
   "MII_Parameters".Connection_Status.opcUaDiagnostics := #Controllers.opcUaDiagnostics.subfunctionStatus;

   // Shift data to display on HMI
   IF #Controllers.opcUaDiagnostics.subfunctionStatus > 65536 THEN
       "MII_Parameters".Connection_Status.aux.opcUaSubfunctionStatus := SHR(IN := #Controllers.opcUaDiagnostics.subfunctionStatus, N := 16);
   END_IF;

   // Output error parameters
   IF NOT #Controllers.opcUaError AND "MII_Parameters".Connection_Status.opcUaConnected THEN
       CASE #Controllers.opcUaStatus OF
           16#0000:
               IF NOT #Controllers.opcUaDone THEN
                   //Client not connected.
                   "MII_Parameters".Connection_Status.aux.diagnosticStatus := 1;
               ELSE
                   //Job successfully executed.
                   "MII_Parameters".Connection_Status.aux.diagnosticStatus := 2;
               END_IF;

           16#7000:
               IF NOT #Controllers.opcUaDone THEN
                   //Client connected and ready for job.
                   "MII_Parameters".Connection_Status.aux.diagnosticStatus := 3;
               ELSE
                   //Connection successfully established and ready for job.
                   "MII_Parameters".Connection_Status.aux.diagnosticStatus := 4;
               END_IF;

           16#7001: //Job is running.
               "MII_Parameters".Connection_Status.aux.diagnosticStatus := 5;
       END_CASE;
   ELSE
       // Output parameters with error
       "MII_Parameters".Connection_Status.aux.diagnosticStatus := #Controllers.opcUaStatus;


   END_IF;
END_REGION

REGION Network 6 (SCL): Try to call method again routine / Not used
   // //Method call timeout
   // #Timers.tryAgain(IN := "MII_Parameters".M000_Status.error,
   //                  PT := t#2s,
   //                  Q => #Auxiliar.tryAgain);

   // IF #Controllers.opcUaConnected AND #Auxiliar.tryAgain THEN
   //              //Try again
   //              IF NOT #CallBuffer[0] THEN
   //                  #CallBuffer[0] := TRUE;

   //                  //Add one attempt to counter
   //                  "MII_Parameters".Connection_Status.aux.nAttemptsTotal := "MII_Parameters".Connection_Status.aux.nAttemptsTotal + 1;
   //              END_IF;

   //              //Restart timer
   //              RESET_TIMER(#Timers.tryAgain);

   //          END_IF;
END_REGION
END_FUNCTION_BLOCK

FUNCTION_BLOCK "0. OpcUaClient"
TITLE = OpcUaClient
{ S7_Optimized_Access := 'TRUE' }
AUTHOR : SiemensAG
VERSION : 1.3
//OPC UA-Client-Wrapper
   VAR_INPUT 
      enable : Bool;   // TRUE: Enable connection to OPC UA server
      read : Bool;   // TRUE: Execute Read functionality
      write : Bool;   // TRUE: Execute Write functionality
      callMethod : Bool;   // TRUE: Execute Method Call
      methodHdlIndex : SInt;   // Index of method in "methodHdls" that should be called
      connectionInfo {InstructionName := 'OPC_UA_SessionConnectInfo'; LibVersion := '1.0'} : OPC_UA_SessionConnectInfo;   // Connection Information for session establishment to OPC UA server
      serverEndpointUrl : String;   // Endpoint of OPC UA server
   END_VAR

   VAR_OUTPUT 
      connected { ExternalWritable := 'False'} : Bool;   // TRUE: Connection to OPC UA server is established and valid
      done { ExternalWritable := 'False'} : Bool;   // TRUE: Functions Read, Write or Method Call were executed successfully
      busy { ExternalWritable := 'False'} : Bool;   // TRUE: FB is working
      error { ExternalWritable := 'False'} : Bool;   // TRUE: FB is in faulty state
      status { ExternalWritable := 'False'} : Word;   // 16#0000 - 16#7FFF: Status of the FB, 16#8000 - 16#FFFF: Error identification
      diagnostics { ExternalWritable := 'False'} : "typeFbDiagnostics";   // Diagnostics information of FB when error occurs
      connectionHdl { ExternalWritable := 'False'} : DWord;   // Connection handle which is used for OPC UA connection to the server
   END_VAR

   VAR_IN_OUT 
      namespaceUris : Variant;   // Pointer to the Namespace URIs of the OPC UA client interface (NULL if not used)
      namespaceIndexes : Variant;   // Pointer to the Namespace Indexes of the OPC UA client interface (NULL if not used)
      readNodeIds : Variant;   // Pointer to the Node-IDs of the nodes to read of the OPC UA client interface (NULL if not used)
      readNodeHdls : Variant;   // Pointer to the Node handles of the registered nodes to read of the OPC UA client interface (NULL if not used)
      readData : Variant;   // Pointer to the storage area for read data (NULL if not used)
      writeNodeIds : Variant;   // Pointer to the Node-IDs of the nodes to write of the OPC UA client interface (NULL if not used)
      writeNodeHdls : Variant;   // Pointer to the Node handles of the registered nodes to write of the OPC UA client interface (NULL if not used)
      writeData : Variant;   // Pointer to the storage area for write data (NULL if not used)
      objNodeIds : Variant;   // Pointer to the Node-IDs of the method objects (instance DB) of the OPC UA client interface (NULL if not used)
      methodNodeIds : Variant;   // Pointer to the Node-IDs of the methods of the OPC UA client Interface (NULL if not used)
      methodHdls : Variant;   // Pointer to the Node handles of the registered methods of the OPC UA client interface (NULL if not used)
      inputArguments : Variant;   // Pointer to the Input Arguments of the called method (NULL if not used)
      outputArguments : Variant;   // Pointer to the Output Arguments of the called method (NULL if not used)
   END_VAR

   VAR 
      instOpcUaConnect {InstructionName := 'OPC_UA_Connect'; LibVersion := '1.0'; ExternalAccessible := 'False'; ExternalVisible := 'False'; ExternalWritable := 'False'} : OPC_UA_Connect;
      instOpcUaConnectionGetStatus {InstructionName := 'OPC_UA_ConnectionGetStatus'; LibVersion := '1.0'; ExternalAccessible := 'False'; ExternalVisible := 'False'; ExternalWritable := 'False'} : OPC_UA_ConnectionGetStatus;
      instOpcUaNamespaceGIL {InstructionName := 'OPC_UA_NamespaceGetIndexList'; LibVersion := '1.0'; ExternalAccessible := 'False'; ExternalVisible := 'False'; ExternalWritable := 'False'} : OPC_UA_NamespaceGetIndexList;
      InstOpcUaGHLRead {InstructionName := 'OPC_UA_NodeGetHandleList'; LibVersion := '1.0'; ExternalAccessible := 'False'; ExternalVisible := 'False'; ExternalWritable := 'False'} : OPC_UA_NodeGetHandleList;
      instOpcUaGHLWrite {InstructionName := 'OPC_UA_NodeGetHandleList'; LibVersion := '1.0'; ExternalAccessible := 'False'; ExternalVisible := 'False'; ExternalWritable := 'False'} : OPC_UA_NodeGetHandleList;
      instOpcUaGHLMethods {InstructionName := 'OPC_UA_MethodGetHandleList'; LibVersion := '1.0'; ExternalAccessible := 'False'; ExternalVisible := 'False'; ExternalWritable := 'False'} : OPC_UA_MethodGetHandleList;   // Get node handles for Methods
      InstOpcUaRHLRead {InstructionName := 'OPC_UA_NodeReleaseHandleList'; LibVersion := '1.0'; ExternalAccessible := 'False'; ExternalVisible := 'False'; ExternalWritable := 'False'} : OPC_UA_NodeReleaseHandleList;
      instOpcUaRHLWrite {InstructionName := 'OPC_UA_NodeReleaseHandleList'; LibVersion := '1.0'; ExternalAccessible := 'False'; ExternalVisible := 'False'; ExternalWritable := 'False'} : OPC_UA_NodeReleaseHandleList;
      instOpcUaRHLMethods {InstructionName := 'OPC_UA_MethodReleaseHandleList'; LibVersion := '1.0'; ExternalAccessible := 'False'; ExternalVisible := 'False'; ExternalWritable := 'False'} : OPC_UA_MethodReleaseHandleList;
      instOpcUaReadList {InstructionName := 'OPC_UA_ReadList'; LibVersion := '1.0'; ExternalAccessible := 'False'; ExternalVisible := 'False'; ExternalWritable := 'False'} : OPC_UA_ReadList;
      instOpcUaWriteList {InstructionName := 'OPC_UA_WriteList'; LibVersion := '1.0'; ExternalAccessible := 'False'; ExternalVisible := 'False'; ExternalWritable := 'False'} : OPC_UA_WriteList;   // Write values of multiple nodes
      instOpcUaMethodCall {InstructionName := 'OPC_UA_MethodCall'; LibVersion := '1.0'; ExternalAccessible := 'False'; ExternalVisible := 'False'; ExternalWritable := 'False'} : OPC_UA_MethodCall;
      instOpcUaDisconnect {InstructionName := 'OPC_UA_Disconnect'; LibVersion := '1.0'; ExternalAccessible := 'False'; ExternalVisible := 'False'; ExternalWritable := 'False'} : OPC_UA_Disconnect;
      statOldTriggers { ExternalAccessible := 'False'; ExternalVisible := 'False'; ExternalWritable := 'False'} : Struct   // Internal structure for Trigger handling
         connect { ExternalAccessible := 'False'; ExternalVisible := 'False'; ExternalWritable := 'False'} : Bool;   // Saved Trigger for Connection establishment
         reconnect { ExternalAccessible := 'False'; ExternalVisible := 'False'; ExternalWritable := 'False'} : Bool;   // Saved Trigger for Connection reestablishment
         disconnect { ExternalAccessible := 'False'; ExternalVisible := 'False'; ExternalWritable := 'False'; S7_SetPoint := 'True'} : Bool;   // Saved Trigger for disconnecting
         read { ExternalAccessible := 'False'; ExternalVisible := 'False'; ExternalWritable := 'False'; S7_SetPoint := 'True'} : Bool;   // Saved Trigger for Read
         write { ExternalAccessible := 'False'; ExternalVisible := 'False'; ExternalWritable := 'False'; S7_SetPoint := 'True'} : Bool;   // Saved Trigger for Write
         callMethod { ExternalAccessible := 'False'; ExternalVisible := 'False'; ExternalWritable := 'False'} : Bool;   // Saved Trigger for Method Call
         clearSession { ExternalAccessible := 'False'; ExternalVisible := 'False'; ExternalWritable := 'False'} : Bool;   // Saved Trigger for Session Clearing
      END_STRUCT;
      statState { ExternalWritable := 'False'} : Int;   // Actual state of the state machine. 0: connect; 1: get Namespaces; 3: Get List Handles; 4: Connected; 5: Disconnect
      statDone { ExternalAccessible := 'False'; ExternalVisible := 'False'; ExternalWritable := 'False'} : Bool;   // Read, Write, MethodCall finished without error.
      statConnected { ExternalAccessible := 'False'; ExternalVisible := 'False'; ExternalWritable := 'False'} : Bool;   // Connection to OPC UA Server is established and valid.
      statBusy { ExternalVisible := 'False'; ExternalWritable := 'False'} : Bool;   // FB is busy.
      statDiagnostics { ExternalAccessible := 'False'; ExternalVisible := 'False'; ExternalWritable := 'False'} : "typeFbDiagnostics";   // Diagnostic structure for internal use.
      statDiagnosticsEmpty { ExternalWritable := 'False'} : "typeFbDiagnostics";   // Empty diagnostic structure, to initialize Output.
      statOpcUaRequests { ExternalAccessible := 'False'; ExternalVisible := 'False'; ExternalWritable := 'False'} : Struct   // Internal structure for OPC UA function blocks requests.
         connect { ExternalAccessible := 'False'; ExternalVisible := 'False'; ExternalWritable := 'False'} : Bool;   // Request for OPC_UA_Connect
         conGS { ExternalAccessible := 'False'; ExternalVisible := 'False'; ExternalWritable := 'False'} : Bool;   // Request for OPC_UA_ConnectionGetStatus
         NGIL { ExternalAccessible := 'False'; ExternalVisible := 'False'; ExternalWritable := 'False'} : Bool;   // Request for OPC_UA_NamespaceGetIndexList
         readGHL { ExternalAccessible := 'False'; ExternalVisible := 'False'; ExternalWritable := 'False'} : Bool;   // Request for OPC_UA_NodeGetHandleList for ReadList
         methodsGHL { ExternalAccessible := 'False'; ExternalVisible := 'False'; ExternalWritable := 'False'} : Bool;   // Request for OPC_UA_MethodGetHandleList
         writeGHL { ExternalAccessible := 'False'; ExternalVisible := 'False'; ExternalWritable := 'False'} : Bool;   // Request for OPC_UA_NodeGetHandleList for WriteList
         read { ExternalAccessible := 'False'; ExternalVisible := 'False'; ExternalWritable := 'False'} : Bool;   // Request for OPC_UA_ReadList
         write { ExternalAccessible := 'False'; ExternalVisible := 'False'; ExternalWritable := 'False'} : Bool;   // Request for OPC_UA_WriteList
         methodCall { ExternalAccessible := 'False'; ExternalVisible := 'False'; ExternalWritable := 'False'} : Bool;   // Request for OPC_UA_MethodCall
         readRHL { ExternalAccessible := 'False'; ExternalVisible := 'False'; ExternalWritable := 'False'} : Bool;   // Request for OPC_UA_NodeReleaseHandleList for ReadList
         writeRHL { ExternalAccessible := 'False'; ExternalVisible := 'False'; ExternalWritable := 'False'} : Bool;   // Request for OPC_UA_NodeReleaseHandleList for WriteList
         methodsRHL { ExternalAccessible := 'False'; ExternalVisible := 'False'; ExternalWritable := 'False'} : Bool;   // Request for OPC_UA_MethodReleaseHandleList
         disconnect { ExternalAccessible := 'False'; ExternalVisible := 'False'; ExternalWritable := 'False'} : Bool;   // Request for OPC_UA_Disconnect
      END_STRUCT;
      statRegisteredLists { ExternalWritable := 'False'} : Struct   // Internal structure for registered Lists/Namespaces. For Diagnostic purpose.
         NamespaceIndexes { ExternalWritable := 'False'} : Bool;   // Namespace Indexes are registered by OPC_UA_NamespaceGetIndexList
         Read { ExternalWritable := 'False'} : Bool;   // Read list is registered by OPC_UA_NodeGetHandleList
         Write { ExternalWritable := 'False'} : Bool;   // Write list is registered by OPC_UA_NodeGetHandleList
         Methods { ExternalWritable := 'False'} : Bool;   // Method list is registered by OPC_UA_MethodGetHandleList
      END_STRUCT;
      statDiagCounter { ExternalWritable := 'False'} : Struct   // Internal structure for counting connects/registrations/functions. For Diagnostic purpose.
         Connect { ExternalVisible := 'False'; ExternalWritable := 'False'} : UInt;   // Counter for successful connects or reconnects.
         NamespaceReg { ExternalWritable := 'False'} : UInt;   // Counter for successful Namespace registrations.
         RegisterRead { ExternalWritable := 'False'} : UInt;   // Counter for successful Read List registrations.
         RegisterWrite { ExternalWritable := 'False'} : UInt;   // Counter for successful Write List registrations.
         RegisterMethods { ExternalWritable := 'False'} : UInt;   // Counter for successful Method List registrations.
         Read { ExternalWritable := 'False'} : UInt;   // Counter for successful Read function executions.
         Write { ExternalWritable := 'False'} : UInt;   // Counter for successful Write function executions.
         MethodCall { ExternalWritable := 'False'} : UInt;   // Counter for successful Method Calls.
      END_STRUCT;
      statMethodResult { ExternalWritable := 'False'} : DWord;   // OPC UA result after Method Call.
      statMethodHdl { ExternalAccessible := 'False'; ExternalVisible := 'False'; ExternalWritable := 'False'} : DWord;   // Calculated Method Handle. Dependend on INPUT: methodHdlIndex.
      statMethodHdlId { ExternalAccessible := 'False'; ExternalVisible := 'False'; ExternalWritable := 'False'} : DInt;   // Internal Variable for INPUT: methodHdlIndex.
      statConnectionHdl { ExternalAccessible := 'False'; ExternalVisible := 'False'; ExternalWritable := 'False'} : DWord;   // Internal Variable for Connection Handle.
      statRHLTrigger { ExternalAccessible := 'False'; ExternalVisible := 'False'; ExternalWritable := 'False'} : Bool;   // Trigger, do start with releasing Lists for disconnect.
      statCheckConnectionStatus { ExternalAccessible := 'False'; ExternalVisible := 'False'; ExternalWritable := 'False'} : Bool;   // If TRUE, OPC_UA_ConnectionGetStatus is called to diagnose the connection.
      statCycDiagTrigger { ExternalAccessible := 'False'; ExternalVisible := 'False'; ExternalWritable := 'False'} : Bool;   // Cyclic trigger for OPC_UA_ConnectionGetStatus-
      instCycDiag {InstructionName := 'IEC_TIMER'; LibVersion := '1.0'; ExternalAccessible := 'False'; ExternalVisible := 'False'; ExternalWritable := 'False'} : IEC_TIMER;   // Timer for cyclic connection diagnostics.
      statOpcUaReadTimeStamps { ExternalWritable := 'False'} : Array[0..#MAX_LIST_LENGTH] of LDT;   // Timestamps of read variables. For diagnostic purpose.
      statSerializeMethodHdls { ExternalAccessible := 'False'; ExternalVisible := 'False'; ExternalWritable := 'False'} : Array[0..1199] of Byte;   // Array for calculating the MethodHdl together with the INPUT methodHdlIndex.
      statOpcUaStatusLists { ExternalWritable := 'False'} : Struct   // Internal structure for Status Lists, that are used by every OPC_UA_xxx FB
         methodRHL { ExternalWritable := 'False'} : Array[0..299] of DWord;   // Status List for Method OPC_UA_ReleaseHandleList
         methodGHL { ExternalWritable := 'False'} : Array[0..299] of DWord;   // Status List for Method OPC_UA_GetHandleList
         writeRHL { ExternalWritable := 'False'} : Array[0..299] of DWord;   // Status List for Write OPC_UA_ReleaseHandleList
         writeList { ExternalWritable := 'False'} : Array[0..299] of DWord;   // Status List for Write OPC_UA_WritedList
         writeGHL { ExternalWritable := 'False'} : Array[0..299] of DWord;   // Status List for WriteOPC_UA_GetHandleList
         readRHL { ExternalWritable := 'False'} : Array[0..299] of DWord;   // Status List for Read OPC_UA_ReleaseHandleList
         readList { ExternalWritable := 'False'} : Array[0..299] of DWord;   // Status List for Read OPC_UA_ReadList
         readGHL { ExternalWritable := 'False'} : Array[0..299] of DWord;   // Status List for Read OPC_UA_GetHandleList
         namespaceGIL { ExternalWritable := 'False'} : Array[0..299] of DWord;   // Status List for Namespace OPC_UA_NamespaceGetIndexList
      END_STRUCT;
   END_VAR

   VAR_TEMP 
      tempIndex : Int;   // Index for finding errors in statOpcUaStatusLists.
      tempRetVal : Int;   // Return value for Serialize function, that is used for calculating statMethodHdl.
      tempConnectTrigger : Bool;   // Temporary trigger for connection establishment.
      tempDisconnectTrigger : Bool;   // Temporary trigger for disconnect.
      tempReadTrigger : Bool;   // Temporary trigger for Read function.
      tempWriteTrigger : Bool;   // Temporary trigger for Write function.
      tempMethodCallTrigger : Bool;   // Temporary trigger for Method Calls.
      tempReconnectTrigger : Bool;   // Temporary trigger for reconnect.
      tempClearSessionTrigger : Bool;   // Temporary trigger for clean up Session.
      tempConnectionHdl : DWord;   // Temporary variable for Connectionhandle hadover after successful connection setup.
   END_VAR

   VAR CONSTANT 
      STATE_CONNECT : Int := 0;   // State for idling until INPUT enable is triggered, to establish a connection.
      STATE_NAMESPACE_GET_INDEX_LIST : Int := 1;   // State for getting Namespace indexes.
      STATE_NODE_GET_HANDLE_LIST : Int := 3;   // State for registration of Read/Write/Method Lists
      STATE_CONNECTED : Int := 4;   // State for idling until INPUT read/write/methodCall has positive edge, to execute function.
      STATE_DISCONNECT : Int := 5;   // State for releasing Read/Write/Method Lists and disconnect.
      CGS_CONNECTED : UDInt := 0;   // OPC_UA_ConnectionGetStatus Connection state is connected.
      CGS_CONN_ERROR : UDInt := 1;   // OPC_UA_ConnectionGetStatus Connection state is in error.
      CGS_SHUTDOWN : UDInt := 2;   // OPC_UA_ConnectionGetStatus Connection state is in shutdown, nodes have to be released and connection terminated.
      CGS_SS_RUNNING : UDInt := 0;   // OPC_UA_ConnectionGetStatus Server state is running.
      CGS_SL_GOOD : Byte := 16#FF;   // OPC_UA_ConnectionGetStatus Connection state is connected.
      STATUS_SESSION_CLEANEDUP : DWord := 16#A000_0105;   // OPC_UA_ConnectionGetStatus: Session is cleaned up and has to be reconnected.
      STATUS_SERVER_NOT_CONNECTED : DWord := 16#800D_0000;   // OPC_UA_ConnectionGetStatus: Choosen Server is not connected.
      STATUS_BAD_CONNECTION_CLOSED : DWord := 16#80AE_0000;   // OPC_UA_ConnectionGetStatus
      STATUS_BAD_INVALID_STATE : DWord := 16#80AF_0000;   // OPC_UA_ConnectionGetStatus: Invalid State of connection. Probably not available anymore.
      STATUS_BUSY : Word := 16#7001;   // Function block is busy.
      STATUS_IDLE : Word := 16#7000;   // Function block idles.
      STATUS_NOT_REGISTERED : Word := 16#80FF;   // Read/Write/Method List is not registered
      STATUS_DONE : Word := 16#0000;   // Read/Write/Method Call was successfully executed.
      CYC_TIME_GCS : Time := T#5S;   // Time for cylic call of OPC_UA_ConnectionGetStatus
      OPC_UA_FUNCTIONS_TIMEOUT : Time := T#10S;   // Timout for all OPC UA Client Function blocks
      ERR_CONNECT : Word := 16#8601;   // Error during connect.
      ERR_NGIL : Word := 16#8602;   // Error during getting Namespace Indexes
      ERR_NGIL_SL : Word := 16#8617;   // Error in Namespace indexes Status list
      ERR_R_GHL : Word := 16#8631;   // Error during Read list registration
      ERR_R_GHL_SL : Word := 16#8731;   // Error in Read handle list Status list
      ERR_W_GHL : Word := 16#8632;   // Error during Write list registration
      ERR_W_GHL_SL : Word := 16#8732;   // Error in Write handle list Status list
      ERR_M_GHL : Word := 16#8633;   // Error during Method list registration
      ERR_M_GHL_SL : Word := 16#8733;   // Error in Method handle List status list
      ERR_RL : Word := 16#8604;   // Error during Read List execution
      ERR_RL_NOTREG : Word := 16#86F4;   // Error, because no Read List is registered, but Read execution was triggered
      ERR_RL_SL : Word := 16#8614;   // Error in Read list status list.
      ERR_WL : Word := 16#8605;   // Error during Write List execution
      ERR_WL_NOTREG : Word := 16#86F5;   // Error, because no Write List is registered, but Write execution was triggered
      ERR_WL_SL : Word := 16#8615;   // Error in Write list status list
      ERR_MC : Word := 16#8606;   // Error durging Method Call execution
      ERR_MC_NOTREG : Word := 16#86F6;   // Error, because no Method List is registered, but Method call execution was triggered
      ERR_MC_SERIALIZE : Word := 16#8616;   // Error during MethodHdl calculation, in Serialize function
      ERR_MC_RESULT : Word := 16#8626;   // Error, that was reported by Methods OPC UA result
      ERR_MC_INDEX_OO_RANGE : Word := 16#8636;
      ERR_R_RHL : Word := 16#8671;   // Error during release of Read List
      ERR_R_RHL_SL : Word := 16#8771;   // Error in Release Read List status list
      ERR_W_RHL : Word := 16#8672;   // Error during realease of Write list
      ERR_W_RHL_SL : Word := 16#8772;   // Error in Release Write List status list
      ERR_M_RHL : Word := 16#8673;   // Error during relaese of Method List
      ERR_M_RHL_SL : Word := 16#8773;   // Error in Release Method List status List
      ERR_DISCON : Word := 16#8608;   // Error during disconnect.
      ERR_CGS : Word := 16#8610;   // Error in OPC_UA_ConnectionGetStatus
      ERR_CGS_CSTATE : Word := 16#8611;   // Error in OPC_UA_ConnectionGetStatus, regarding Connection Status
      ERR_CGS_CSTATE_SHUTDOWN : Word := 16#8711;   // Error in OPC_UA_ConnectionGetStats, Connection was shut down
      ERR_CGS_SSTATE : Word := 16#8612;   // Error in OPC_UA_ConnectionGetStatus, regarding Server State
      ERR_CGS_SLVL : Word := 16#8613;   // Error in OPC_UA_ConnectionGetStatus, regarding Service Level
      MAX_LIST_LENGTH : UInt := 299;   // Maximum lenth of Write/Readlist
      MAX_LENGTH_METHOD_INDEX : Int := 99;   // maximum length of MethodHdls (max 100 Methods per MethodList)
   END_VAR


BEGIN
	//=============================================================================
	// Siemens AG (c)Copyright (2019)
	//-----------------------------------------------------------------------------
	// Library: -
	// Tested with: CPU 1516-3 PN/DP;  FW 2.9
	// Engineering: TIA Portal (V16)
	// Restrictions: -
	// Requirements: OPC UA Client activated, Fimware V2.8; Set PLC time
	// Functionality: Encapsulates OPC UA client blocks for read, write and method
	//                call including connection handling and diagnosis
	//-----------------------------------------------------------------------------
	// Change log table:
	// Version    Date         Expert in charge           Changes applied
	// 01.00.00   01.02.2019   Siemens SUP Applications   First released version
	// 01.01.00   31.11.2019   Siemens SUP Applications   Interface, Styleguide and user program performance changes
	// 01.02.00   15.10.2020   Siemens SUP Applications   Bugfixes
	// 01.03.00   28.07.2021   Siemens SUP Applications   Fixed RHL issues
	// 01.04.00   10.11.2022   Siemens SUP Applications   Fixed RHL issues and stabilization of errorhandling
	//=============================================================================
	
	
	//State machine
	CASE #statState OF
	  #STATE_CONNECT:
	    REGION Connection Handling
	      //initialize FB
	      IF NOT #enable THEN
	        #statBusy := FALSE;
	        #statDone := FALSE;
	        #statDiagnostics := #statDiagnosticsEmpty;
	        #statOldTriggers.connect := FALSE;
	        #statConnected := FALSE;
	        #statDiagnostics.status := #STATUS_DONE;
	        #statCheckConnectionStatus := FALSE;
	        #statOpcUaRequests.conGS := FALSE;
	      END_IF;
	      
	      //Rising Edge detection of connect
	      #tempConnectTrigger := #enable AND NOT #statOldTriggers.connect;
	      #statOldTriggers.connect := #enable;
	      //Rising Edge detection for Reconnect functionality
	      #tempReconnectTrigger := #enable AND NOT #statConnected
	      AND #statDiagnostics.subfunctionStatus = UDINT_TO_DWORD(#CGS_SHUTDOWN)
	      AND NOT #statOldTriggers.reconnect;
	      #statOldTriggers.reconnect := #enable AND NOT #statConnected
	      AND #statDiagnostics.subfunctionStatus = UDINT_TO_DWORD(#CGS_SHUTDOWN);
	      
	      //If Connect requested, start connection establishment
	      //---------CONNECT HANDLING-------------
	      //--------------------------------------
	      IF #tempConnectTrigger OR #tempReconnectTrigger THEN
	        IF #statConnectionHdl = 16#0 THEN
	          // no connectionHdl is used -> ready to connect
	          #statOpcUaRequests.connect := TRUE;
	          // set FB outputs
	          #statBusy := TRUE;
	          #statDiagnostics.status := #STATUS_BUSY;
	        ELSE
	          //connectionHdl might be defect, first delete connectionHdl
	          //-> not ready to connect
	          #statOpcUaRequests.disconnect := TRUE;
	          //set FB Outputs
	          #statBusy := TRUE;
	          #statDiagnostics.status := #STATUS_BUSY;
	        END_IF;
	      ELSE
	        IF #instOpcUaDisconnect.Error OR #instOpcUaDisconnect.Done AND #enable THEN
	          //possibly open connection handle is not available or is disconnected
	          //-> ready to connect
	          #statOpcUaRequests.disconnect := FALSE;
	          #statOpcUaRequests.connect := TRUE;
	          #statConnectionHdl := 0;
	        ELSE
	          //nothing done by OPC UA Disconnect block -> Not ready to connect
	          #statOpcUaRequests.connect := FALSE;
	        END_IF;
	      END_IF;
	      
	      //Error at connection establishment
	      IF #instOpcUaConnect.Error THEN
	        #statDone := FALSE;
	        #statConnected := FALSE;
	        #statDiagnostics.status := #ERR_CONNECT;
	        #statDiagnostics.subfunctionStatus := #instOpcUaConnect.Status;
	      END_IF;
	      
	      //Connection establishment was successful
	      IF #instOpcUaConnect.Done THEN
	        #statConnected := TRUE;
	        #statOldTriggers.reconnect := FALSE;
	        #statDiagCounter.Connect += 1;
	        #statState := #STATE_NAMESPACE_GET_INDEX_LIST;
	      END_IF;
	      
	    END_REGION
	    
	  #STATE_NAMESPACE_GET_INDEX_LIST:
	    REGION Handle Namespaces
	      //Request Namespace get Indexlist
	      #statOpcUaRequests.NGIL := TRUE;
	      #statDiagnostics.status := #STATUS_BUSY;
	      
	      // Get Index List was not successful
	      IF #instOpcUaNamespaceGIL.Error THEN
	        //--> Call ConnectionGetStatus if Status = "16#800D0000"
	        IF #instOpcUaNamespaceGIL.Status = #STATUS_SERVER_NOT_CONNECTED THEN
	          #statCheckConnectionStatus := TRUE;
	        ELSE
	          #statState := #STATE_CONNECT;
	        END_IF;
	        #statOpcUaRequests.NGIL := FALSE;
	        // => OUT
	        #statBusy := FALSE;
	        #statDiagnostics.status := #ERR_NGIL;
	        #statDiagnostics.subfunctionStatus := #instOpcUaNamespaceGIL.Status;
	      END_IF;
	      
